// Mitsubishi GX Works2 project: BookEX6_48 Network   PLC: Q13UDV

// global labels: QPLCSpecial
VAR_GLOBAL
  sbGetTime AT SM213 : BOOL;
  sbOn AT SM400 : BOOL;
  sbOff AT SM401 : BOOL;
  sbOn1Time AT SM402 : BOOL;
  sbOff1Time AT SM403 : BOOL;
  sb5ms AT SM409 : BOOL;
  sdSwitch AT SD200 : INT;
  sdTime03 AT SD212 : INT;
  sdTime04 AT SD213 : INT;
  sdTime02 AT SD211 : INT;
  sdTime01 AT SD210 : INT;
  sdScanTime1 AT SD521 : INT;
  sdScanTimeMin1 AT SD525 : INT;
  sdScanTimeMin AT SD524 : INT;
  sdScanTimeMax1 AT SD527 : INT;
  sdScanTimeMax AT SD526 : INT;
  sbErrInfo2 AT SM16 : BOOL;
  sbErrInfo AT SM5 : BOOL;
  sbSelfError AT SM1 : BOOL;
  sbDiagError AT SM0 : BOOL;
  sbResetErr AT SM50 : BOOL;
  sbSetTime AT SM210 : BOOL;
  sbFuse AT SM60 : BOOL;
  sbOpError AT SM56 : BOOL;
  sbPowerDown AT SM53 : BOOL;
  sbBatLow AT SM52 : BOOL;
  sbBatLowL AT SM51 : BOOL;
  sbSTOP AT SM203 : BOOL;
  sbPAUSE AT SM204 : BOOL;
  sbNsec AT SM414 : BOOL;
  sb1000ms AT SM413 : BOOL;
  sb500ms AT SM412 : BOOL;
  sbNms AT SM415 : BOOL;
  sbUserClk4 AT SM424 : BOOL;
  sbUserClk3 AT SM423 : BOOL;
  sbUserClk2 AT SM422 : BOOL;
  sbUserClk1 AT SM421 : BOOL;
  sbUserClk0 AT SM420 : BOOL;
  sdBatLowL AT SD51 : INT;
  sdPLCErrInfo AT SD4 : INT;
  sdPLCErrDate2 AT SD3 : INT;
  sdPLCErrDate1 AT SD2 : INT;
  sdPLCErrDate0 AT SD1 : INT;
  sdPLCErrCode AT SD0 : INT;
  sdFuse AT SD60 : INT;
  sdPowerDown AT SD53 : INT;
  sdBatLow AT SD52 : INT;
  sdCPUSts AT SD203 : INT;
  sdLed AT SD201 : INT;
  sdScanTime AT SD520 : INT;
  sdCntNsec AT SD414 : INT;
  sdCnt1sec AT SD412 : INT;
  sdCntScan AT SD420 : INT;
  sdCntNms AT SD415 : INT;
  sb100ms AT SM411 : BOOL;
  sb50ms AT SM410 : BOOL;
  sdSckOpenComp AT SD1282 : WORD;
  sdSckOpenReq AT SD1284 : WORD;
  sdSckDataRx AT SD1286 : WORD;
  sdSckConn AT SD1288 : WORD;
END_VAR

// global labels: Network
VAR_GLOBAL
  aSendData1 AT D100 : ARRAY [0..4] OF INT;
  aiTxData AT D4000 : ARRAY [0..99] OF INT;
  aiRxData AT D4100 : ARRAY [0..99] OF INT;
  iOpenOK AT D3900 : INT;
  iOpenERR AT D3901 : INT;
  iSendOK AT D3902 : INT;
  iSendERR AT D3903 : INT;
  iCloseOK AT D3906 : INT;
  iCloseERR AT D3907 : INT;
  iRecvOK AT D3904 : INT;
  iRecvERR AT D3905 : INT;
  aiTxData2 AT D4200 : ARRAY [0..99] OF INT;
  aiRxData2 AT D4300 : ARRAY [0..99] OF INT;
  iOpenOK2 AT D3908 : INT;
  iOpenERR2 AT D3909 : INT;
  iSendOK2 AT D3910 : INT;
  iSendERR2 AT D3911 : INT;
  iRecvOK2 AT D3912 : INT;
  iRecvERR2 AT D3913 : INT;
  iCloseOK2 AT D3914 : INT;
  iCloseERR2 AT D3915 : INT;
  iEOpenComp AT D3916 : INT;
  iEOpenReq AT D3917 : INT;
  iERecvFlag AT D3918 : INT;
  iOpenCode AT D3919 : INT;
  iSendCode AT D3920 : INT;
  iRecvCode AT D3921 : INT;
  iCloseCode AT D3922 : INT;
  iOpenCode2 AT D3923 : INT;
  iSendCode2 AT D3924 : INT;
  iRecvCode2 AT D3925 : INT;
  iCloseCode2 AT D3926 : INT;
  aRecvData1 AT D105 : ARRAY [0..4] OF INT;
  aSendData2 AT D110 : ARRAY [0..4] OF INT;
  aRecvData2 AT D115 : ARRAY [0..4] OF INT;
  aSendData3 AT D120 : ARRAY [0..4] OF INT;
  aRecvData3 AT D125 : ARRAY [0..4] OF INT;
  aRdata AT D140 : ARRAY [0..9] OF INT;
  aSLMPDataTx AT D150 : ARRAY [0..9] OF WORD;
  aSLMPDataRx AT D160 : ARRAY [0..9] OF WORD;
END_VAR

// global labels: Global
VAR_GLOBAL
  bVar0 AT M5000 : BOOL;
  abArray0 AT M5010 : ARRAY [0..49] OF BOOL;
  sStr0 AT D5000 : STRING[199];
  sStr1 AT D5100 : STRING[199];
  sStr2 AT D5200 : STRING[199];
  sStr3 AT D5300 : STRING[199];
  sStr4 AT D5400 : STRING[199];
  sStr5 AT D5500 : STRING[199];
  sStr6 AT D5600 : STRING[199];
  sStr7 AT D5700 : STRING[199];
  sStr8 AT D5800 : STRING[199];
  sStr9 AT D5900 : STRING[199];
  iVar0 AT D4500 : INT;
  iVar1 AT D4501 : INT;
  iVar2 AT D4502 : INT;
  iVar3 AT D4503 : INT;
  iVar4 AT D4504 : INT;
  iVar5 AT D4505 : INT;
  iVar6 AT D4506 : INT;
  iVar7 AT D4507 : INT;
  iVar8 AT D4508 : INT;
  iVar9 AT D4509 : INT;
  dVar0 AT D4510 : DINT;
  dVar1 AT D4512 : DINT;
  dVar2 AT D4514 : DINT;
  dVar3 AT D4516 : DINT;
  dVar4 AT D4518 : DINT;
  dVar5 AT D4520 : DINT;
  dVar6 AT D4522 : DINT;
  dVar7 AT D4524 : DINT;
  dVar8 AT D4526 : DINT;
  dVar9 AT D4528 : DINT;
  wVar0 AT D4530 : WORD;
  wVar1 AT D4531 : WORD;
  wVar2 AT D4532 : WORD;
  wVar3 AT D4533 : WORD;
  wVar4 AT D4534 : WORD;
  wVar5 AT D4535 : WORD;
  wVar6 AT D4536 : WORD;
  wVar7 AT D4537 : WORD;
  wVar8 AT D4538 : WORD;
  wVar9 AT D4539 : WORD;
  dwVar0 AT D4540 : DWORD;
  dwVar1 AT D4542 : DWORD;
  dwVar2 AT D4544 : DWORD;
  dwVar3 AT D4546 : DWORD;
  dwVar4 AT D4548 : DWORD;
  dwVar5 AT D4550 : DWORD;
  dwVar6 AT D4552 : DWORD;
  dwVar7 AT D4554 : DWORD;
  dwVar8 AT D4556 : DWORD;
  dwVar9 AT D4558 : DWORD;
  fsVar0 AT D4560 : REAL;
  fsVar1 AT D4562 : REAL;
  fsVar2 AT D4564 : REAL;
  fsVar3 AT D4566 : REAL;
  fsVar4 AT D4568 : REAL;
  fsVar5 AT D4570 : REAL;
  fsVar6 AT D4572 : REAL;
  fsVar7 AT D4574 : REAL;
  fsVar8 AT D4576 : REAL;
  fsVar9 AT D4578 : REAL;
  fdVar0 AT D4580 : LREAL;
  tTime0 AT D4620 : TIME;
  tTime1 AT D4622 : TIME;
  tTime2 AT D4624 : TIME;
  tTime3 AT D4626 : TIME;
  tTime4 AT D4628 : TIME;
  tTime5 AT D4630 : TIME;
  tTime6 AT D4632 : TIME;
  tTime7 AT D4634 : TIME;
  tTime8 AT D4636 : TIME;
  tTime9 AT D4638 : TIME;
  tTime10 AT D4640 : TIME;
  bVar1 AT M5001 : BOOL;
  bVar2 AT M5002 : BOOL;
  bVar3 AT M5003 : BOOL;
  bVar4 AT M5004 : BOOL;
  bVar5 AT M5005 : BOOL;
  bVar6 AT M5006 : BOOL;
  bVar7 AT M5007 : BOOL;
  bVar8 AT M5008 : BOOL;
  bVar9 AT M5009 : BOOL;
  abArray1 AT M5060 : ARRAY [0..49] OF BOOL;
  abArray2 AT M5110 : ARRAY [0..49] OF BOOL;
  abArray3 AT M5160 : ARRAY [0..49] OF BOOL;
  abArray4 AT M5210 : ARRAY [0..49] OF BOOL;
  abArray5 AT M5260 : ARRAY [0..49] OF BOOL;
  abArray6 AT M5310 : ARRAY [0..49] OF BOOL;
  abArray7 AT M5360 : ARRAY [0..49] OF BOOL;
  abArray8 AT M5410 : ARRAY [0..49] OF BOOL;
  abArray9 AT M5460 : ARRAY [0..49] OF BOOL;
  fdVar1 AT D4584 : LREAL;
  fdVar2 AT D4588 : LREAL;
  fdVar3 AT D4592 : LREAL;
  fdVar4 AT D4596 : LREAL;
  fdVar5 AT D4600 : LREAL;
  fdVar6 AT D4604 : LREAL;
  fdVar7 AT D4608 : LREAL;
  fdVar8 AT D4612 : LREAL;
  fdVar9 AT D4616 : LREAL;
  afsPen0 AT D2000 : ARRAY [0..499] OF REAL;
  afsPen1 AT D3000 : ARRAY [0..499] OF REAL;
END_VAR
// user libraries (not included): HMI

PROGRAM ExEpasCact
VAR
  bOpenReqC : BOOL;
  bOpenOkC : BOOL;
  bOpenErrC : BOOL;
  abOpenResC : ARRAY [0..1] OF BOOL;
  acOpenData : ARRAY [0..9] OF INT;
  bSendReqC : BOOL;
  bSendOkC : BOOL;
  bSendErrC : BOOL;
  abSendResC : ARRAY [0..1] OF BOOL;
  acSendDataC : ARRAY [0..1] OF INT;
  bRecvOkC : BOOL;
  bRecvErrC : BOOL;
  abRecvResC : ARRAY [0..1] OF BOOL;
  bCloseReq : BOOL;
  bCloseOkC : BOOL;
  bCloseErrC : BOOL;
  abCloseResC : ARRAY [0..1] OF BOOL;
  acCloseData : ARRAY [0..1] OF INT;
  CntSend1 : INT;
  CntSend2 : INT;
  CntRecv1 : INT;
  CntRecv2 : INT;
  Mov4INT_1 : Mov4INT;
  Mov8INT_1 : Mov8INT;
  acRdCtrl : ARRAY [0..9] OF INT;
  Mov4INT_2 : Mov4INT;
  bOpenReqE : BOOL;
  bOpenOkE : BOOL;
  bOpenErrE : BOOL;
  abOpenResE : ARRAY [0..1] OF BOOL;
  bSendErrE : BOOL;
  bSendOkE : BOOL;
  bSendReqE : BOOL;
  abSendResE : ARRAY [0..1] OF BOOL;
  abRecvResE : ARRAY [0..1] OF BOOL;
  bRecvErrE : BOOL;
  bRecvOkE : BOOL;
  abCloseResE : ARRAY [0..1] OF BOOL;
  bCloseErrE : BOOL;
  bCloseOkE : BOOL;
  acSendDataE : ARRAY [0..1] OF INT;
  acRecvDataC : ARRAY [0..1] OF INT;
  acRecvDataE : ARRAY [0..1] OF INT;
  Word2Bit8_1 : Word2Bit8;
  Word2Bit8_2 : Word2Bit8;
  Word2Bit8_3 : Word2Bit8;
  Word2Bit8_4 : Word2Bit8;
  Word2Bit8_5 : Word2Bit8;
  Word2Bit8_6 : Word2Bit8;
  ErrCodeSC : INT;
  ErrCodeSE : INT;
  Mov4INT_3 : Mov4INT;
  bChangeReqC : BOOL;
  Mov4INT_4 : Mov4INT;
  acRmodeData : ARRAY [0..3] OF INT;
  TON_1 : TON;
  CntRecvErr1 : INT;
  CntRecvErr2 : INT;
  TON_2 : TON;
  ErrCodeRC : INT;
  ErrCodeRE : INT;
  bModeReq : BOOL;
  acRdata : ARRAY [0..1] OF INT;
END_VAR
(* structured ladder/FBD written out as ST: instructions are called as NAME(EN, inputs, outputs); _pN, _eN, _tN stand for wires *)
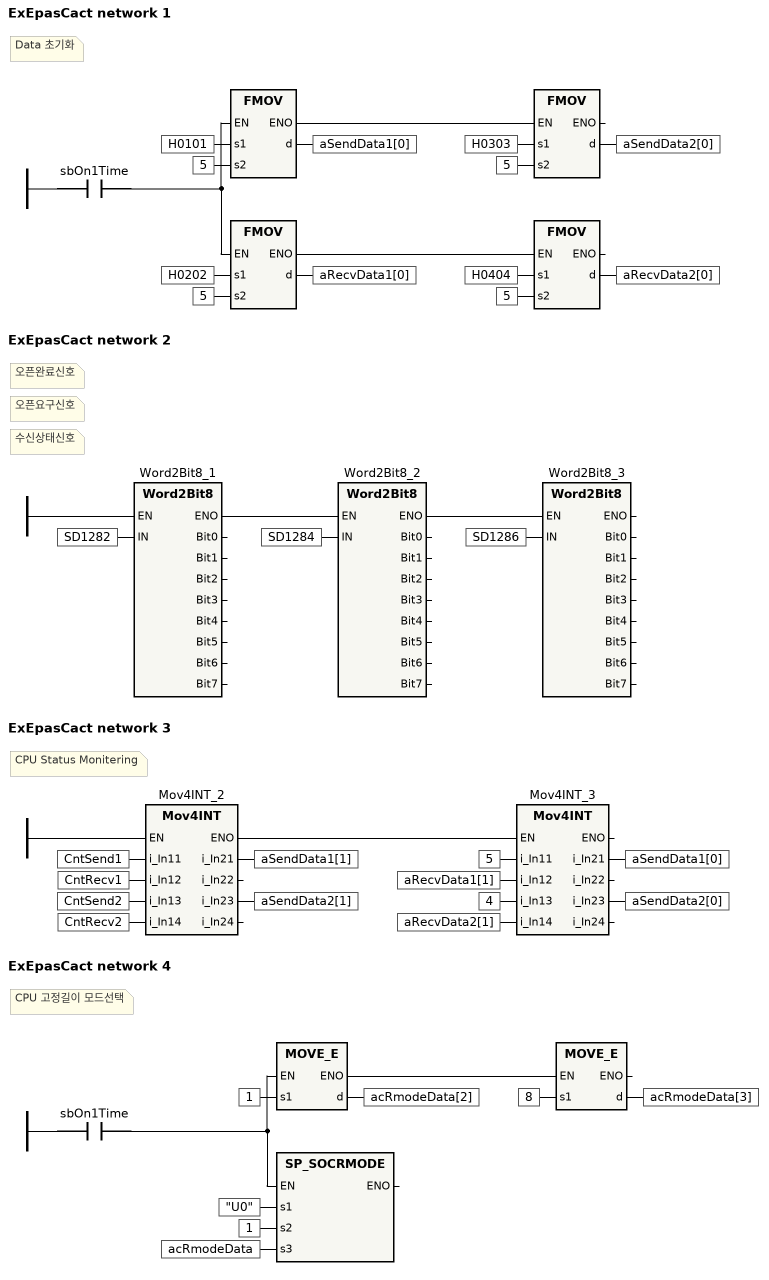
(* network 1 *)
(* Data 초기화 *)
_e1 := FMOV(sbOn1Time, H0101, 5, aSendData1[0]);
FMOV(_e1, H0303, 5, aSendData2[0]);
_e2 := FMOV(sbOn1Time, H0202, 5, aRecvData1[0]);
FMOV(_e2, H0404, 5, aRecvData2[0]);
(* network 2 *)
(* 오픈완료신호 *)
(* 오픈요구신호 *)
(* 수신상태신호 *)
Word2Bit8_1(EN := TRUE, IN := SD1282);
Word2Bit8_2(EN := Word2Bit8_1.ENO, IN := SD1284);
Word2Bit8_3(EN := Word2Bit8_2.ENO, IN := SD1286);
(* network 3 *)
(* CPU Status Monitering *)
Mov4INT_2(EN := TRUE, i_In11 := CntSend1, i_In12 := CntRecv1, i_In13 := CntSend2, i_In14 := CntRecv2, i_In21 => aSendData1[1], i_In23 => aSendData2[1]);
Mov4INT_3(EN := Mov4INT_2.ENO, i_In11 := 5, i_In12 := aRecvData1[1], i_In13 := 4, i_In14 := aRecvData2[1], i_In21 => aSendData1[0], i_In23 => aSendData2[0]);
(* network 4 *)
(* CPU 고정길이 모드선택 *)
_e1 := MOVE_E(sbOn1Time, 1, acRmodeData[2]);
MOVE_E(_e1, 8, acRmodeData[3]);
SP_SOCRMODE(sbOn1Time, "U0", 1, acRmodeData);
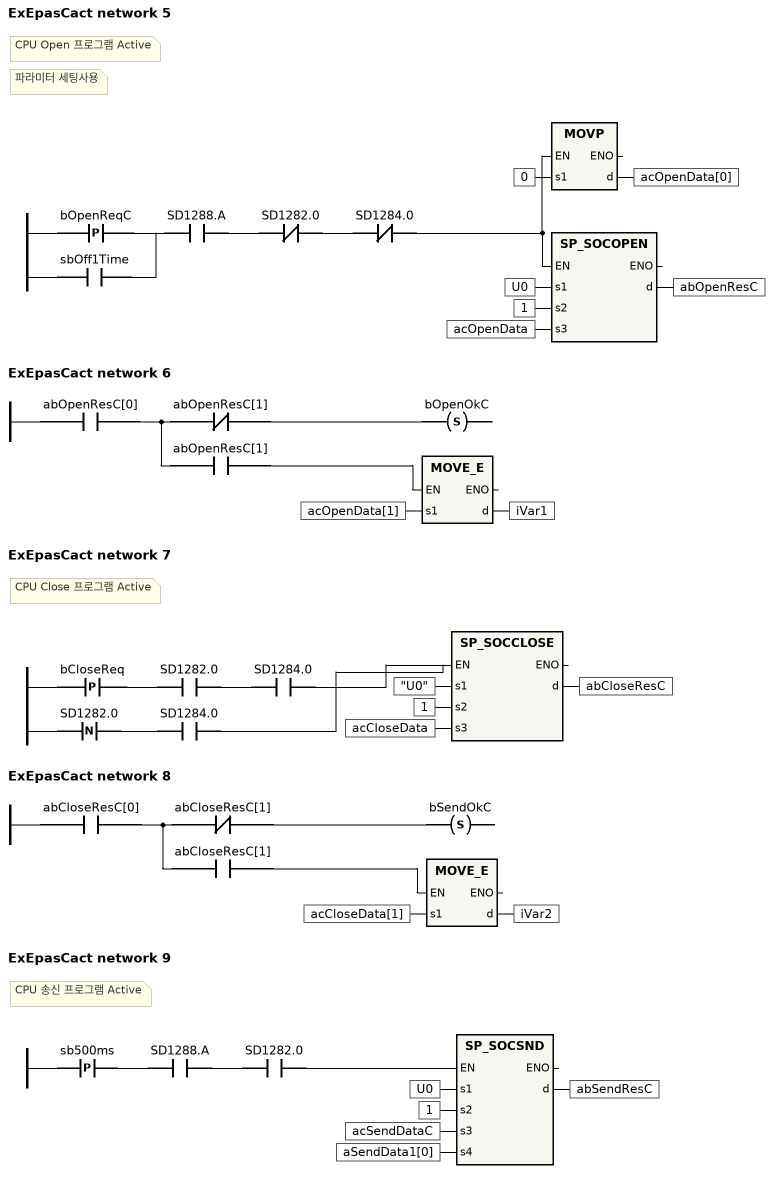
(* network 5 *)
(* CPU Open 프로그램 Active *)
(* 파라미터 세팅사용 *)
_p1 := (((LDP(TRUE, bOpenReqC) OR sbOff1Time) AND SD1288.A) AND NOT SD1282.0) AND NOT SD1284.0;
MOVP(_p1, 0, acOpenData[0]);
SP_SOCOPEN(_p1, U0, 1, acOpenData, abOpenResC);
(* network 6 *)
SET(abOpenResC[0] AND NOT abOpenResC[1], bOpenOkC);
MOVE_E(abOpenResC[0] AND abOpenResC[1], acOpenData[1], iVar1);
(* network 7 *)
(* CPU Close 프로그램 Active *)
SP_SOCCLOSE((LDP(TRUE, bCloseReq) AND SD1282.0 AND SD1284.0) OR (LDF(TRUE, SD1282.0) AND SD1284.0), "U0", 1, acCloseData, abCloseResC);
(* network 8 *)
SET(abCloseResC[0] AND NOT abCloseResC[1], bSendOkC);
MOVE_E(abCloseResC[0] AND abCloseResC[1], acCloseData[1], iVar2);
(* network 9 *)
(* CPU 송신 프로그램 Active *)
SP_SOCSND(LDP(TRUE, sb500ms) AND SD1288.A AND SD1282.0, U0, 1, acSendDataC, aSendData1[0], abSendResC);
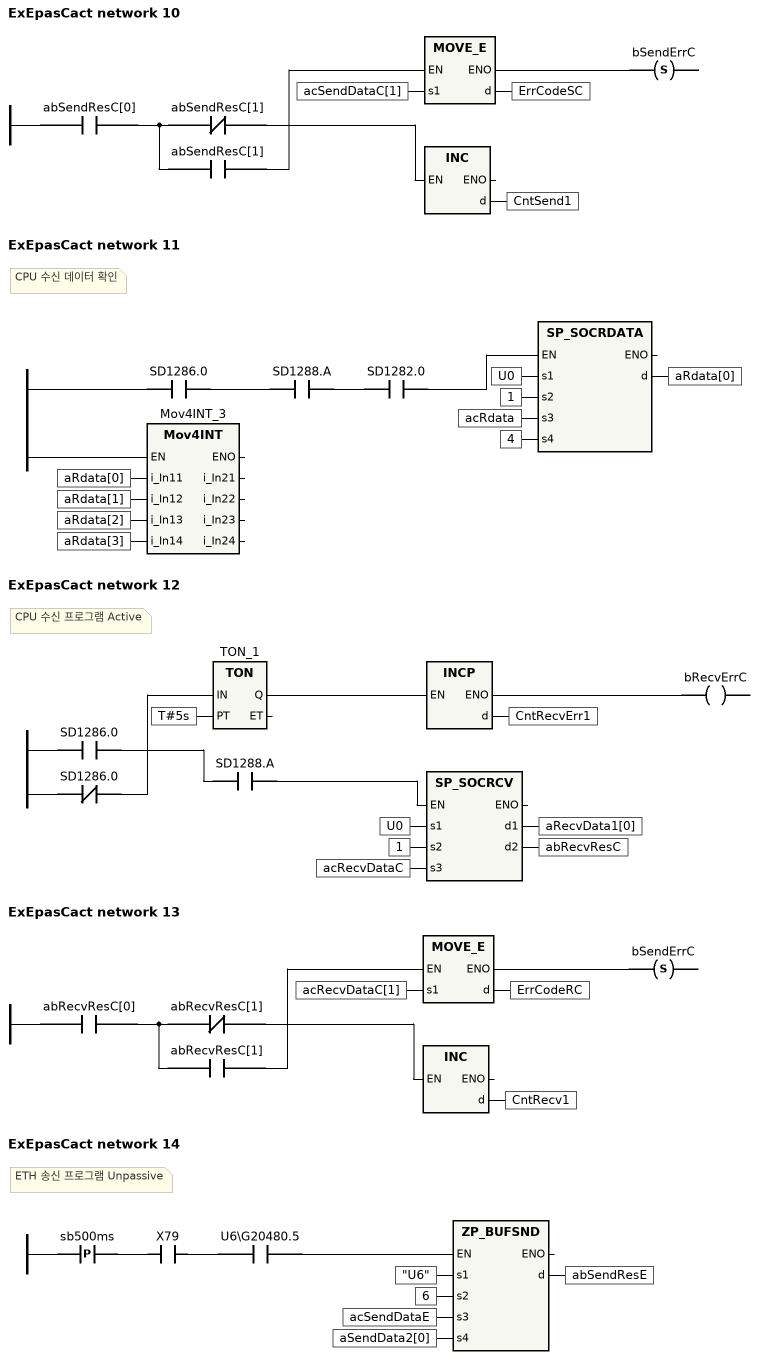
(* network 10 *)
INC(abSendResC[0] AND NOT abSendResC[1], CntSend1);
_e1 := MOVE_E(abSendResC[0] AND abSendResC[1], acSendDataC[1], ErrCodeSC);
SET(_e1, bSendErrC);
(* network 11 *)
(* CPU 수신 데이터 확인 *)
SP_SOCRDATA(SD1286.0 AND SD1288.A AND SD1282.0, U0, 1, acRdata, 4, aRdata[0]);
Mov4INT_3(EN := TRUE, i_In11 := aRdata[0], i_In12 := aRdata[1], i_In13 := aRdata[2], i_In14 := aRdata[3]);
(* network 12 *)
(* CPU 수신 프로그램 Active *)
SP_SOCRCV(SD1286.0 AND SD1288.A, U0, 1, acRecvDataC, aRecvData1[0], abRecvResC);
TON_1(IN := NOT SD1286.0, PT := T#5s);
_e1 := INCP(TON_1.Q, CntRecvErr1);
bRecvErrC := _e1;
(* network 13 *)
INC(abRecvResC[0] AND NOT abRecvResC[1], CntRecv1);
_e1 := MOVE_E(abRecvResC[0] AND abRecvResC[1], acRecvDataC[1], ErrCodeRC);
SET(_e1, bSendErrC);
(* network 14 *)
(* ETH 송신 프로그램 Unpassive *)
ZP_BUFSND(LDP(TRUE, sb500ms) AND X79 AND U6\G20480.5, "U6", 6, acSendDataE, aSendData2[0], abSendResE);
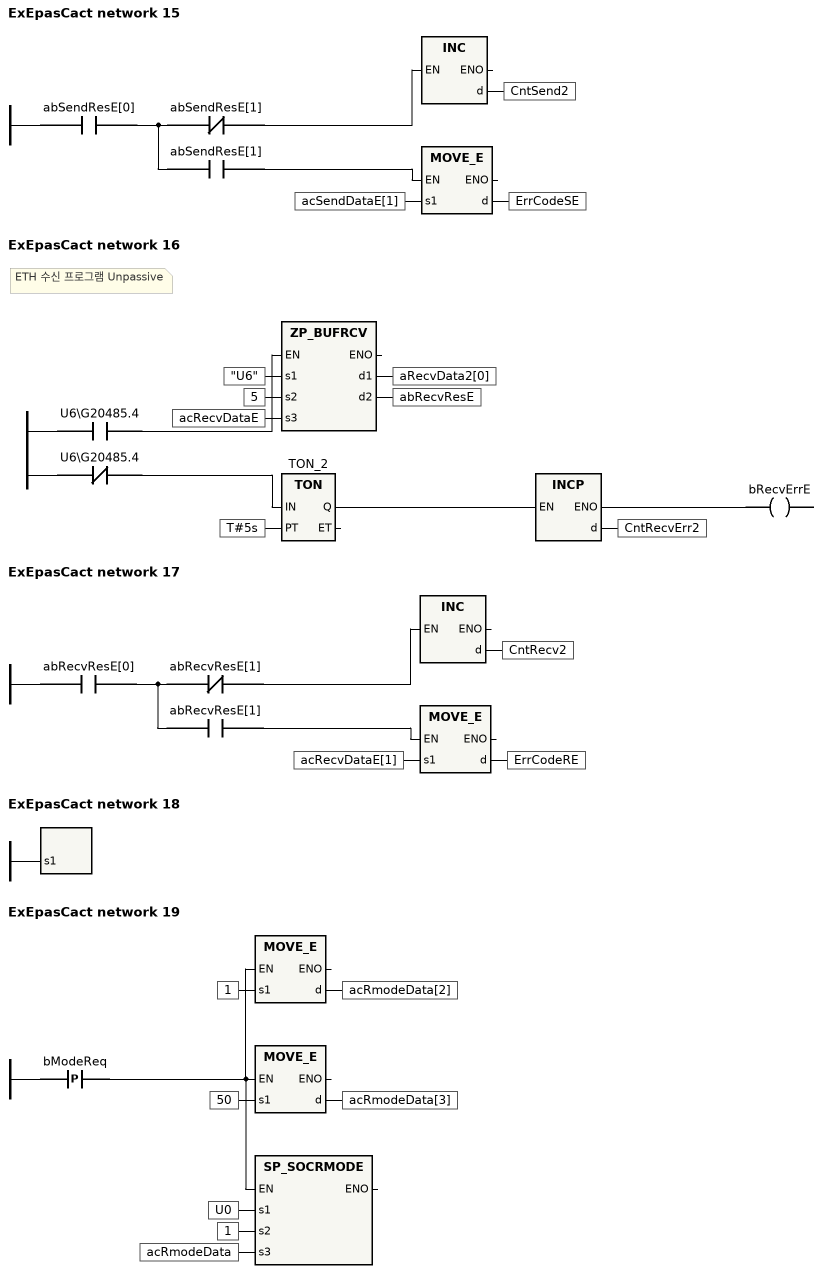
(* network 15 *)
INC(abSendResE[0] AND NOT abSendResE[1], CntSend2);
MOVE_E(abSendResE[0] AND abSendResE[1], acSendDataE[1], ErrCodeSE);
(* network 16 *)
(* ETH 수신 프로그램 Unpassive *)
ZP_BUFRCV(U6\G20485.4, "U6", 5, acRecvDataE, aRecvData2[0], abRecvResE);
TON_2(IN := NOT U6\G20485.4, PT := T#5s);
_e1 := INCP(TON_2.Q, CntRecvErr2);
bRecvErrE := _e1;
(* network 17 *)
INC(abRecvResE[0] AND NOT abRecvResE[1], CntRecv2);
MOVE_E(abRecvResE[0] AND abRecvResE[1], acRecvDataE[1], ErrCodeRE);
(* network 18 *)
(* element kind 10  <- TRUE *)
(* network 19 *)
_p1 := LDP(TRUE, bModeReq);
MOVE_E(_p1, 1, acRmodeData[2]);
MOVE_E(_p1, 50, acRmodeData[3]);
SP_SOCRMODE(_p1, U0, 1, acRmodeData);
END_PROGRAM

PROGRAM xEx_ethOPENact
(* structured ladder/FBD written out as ST: instructions are called as NAME(EN, inputs, outputs); _pN, _eN, _tN stand for wires *)
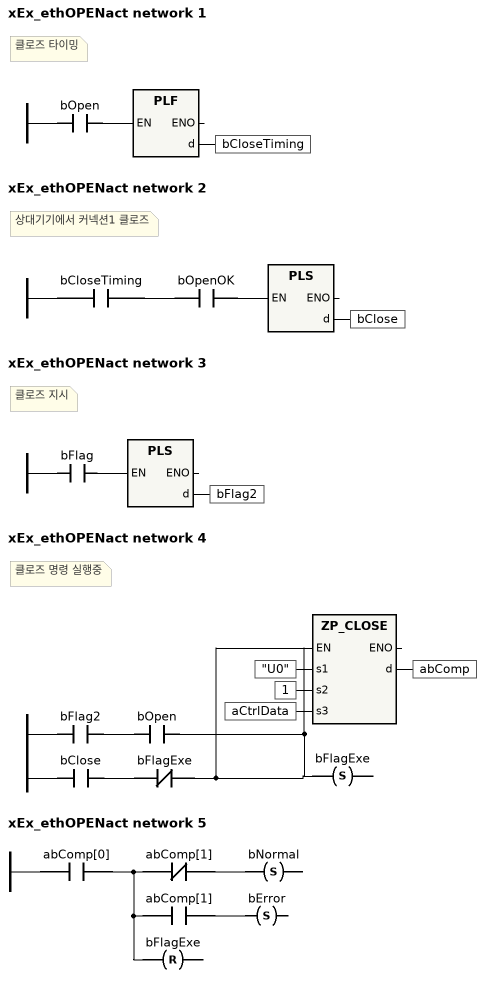
(* network 1 *)
(* 클로즈 타이밍 *)
PLF(bOpen, bCloseTiming);
(* network 2 *)
(* 상대기기에서 커넥션1 클로즈 *)
PLS(bCloseTiming AND bOpenOK, bClose);
(* network 3 *)
(* 클로즈 지시 *)
PLS(bFlag, bFlag2);
(* network 4 *)
(* 클로즈 명령 실행중 *)
_p1 := (bFlag2 AND bOpen) OR (bClose AND NOT bFlagExe);
ZP_CLOSE(_p1, "U0", 1, aCtrlData, abComp);
SET(_p1, bFlagExe);
(* network 5 *)
SET(abComp[0] AND NOT abComp[1], bNormal);
SET(abComp[0] AND abComp[1], bError);
RST(abComp[0], bFlagExe);
END_PROGRAM

PROGRAM xEx_OPENact
VAR
  Mov4INT_1 : Mov4INT;
  abOpenComp : ARRAY [0..1] OF BOOL;
  acOpenData : ARRAY [0..9] OF INT;
  abSendComp : ARRAY [0..1] OF BOOL;
  acSendData : ARRAY [0..1] OF INT;
  abRecvComp : ARRAY [0..1] OF BOOL;
  acRecvData : ARRAY [0..1] OF INT;
  abCloseComp : ARRAY [0..1] OF BOOL;
  acCloseData : ARRAY [0..1] OF INT;
  Word2Bit_1 : Word2Bit;
  Word2Bit_2 : Word2Bit;
  Word2Bit_3 : Word2Bit;
  abOpen : ARRAY [1..16] OF BOOL;
  abReq : ARRAY [1..16] OF BOOL;
  abRecv : ARRAY [1..16] OF BOOL;
  abOpenComp2 : ARRAY [0..1] OF BOOL;
  acOpenData2 : ARRAY [0..9] OF INT;
  abSendComp2 : ARRAY [0..1] OF BOOL;
  acSendData2 : ARRAY [0..1] OF INT;
  abRecvComp2 : ARRAY [0..1] OF BOOL;
  acRecvData2 : ARRAY [0..1] OF INT;
  abCloseComp2 : ARRAY [0..1] OF BOOL;
  acCloseData2 : ARRAY [0..1] OF INT;
  Mov4INT_2 : Mov4INT;
  Word2Bit_4 : Word2Bit;
  Word2Bit_5 : Word2Bit;
  Word2Bit_6 : Word2Bit;
  abRecv2 : ARRAY [1..16] OF BOOL;
  abOpen2 : ARRAY [1..16] OF BOOL;
  abReq2 : ARRAY [1..16] OF BOOL;
  bRecvOK : BOOL;
END_VAR
(* structured ladder/FBD written out as ST: instructions are called as NAME(EN, inputs, outputs); _pN, _eN, _tN stand for wires *)
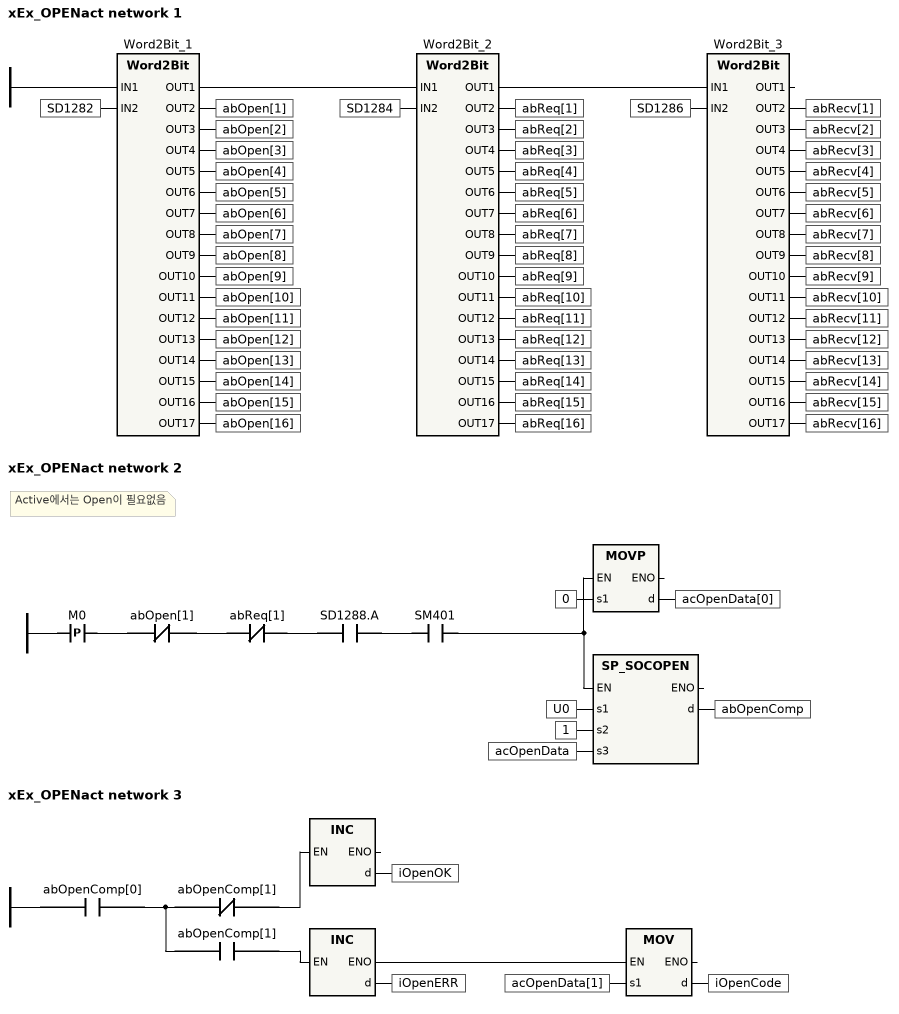
(* network 1 *)
Word2Bit_1(IN1 := TRUE, IN2 := SD1282, OUT2 => abOpen[1], OUT3 => abOpen[2], OUT4 => abOpen[3], OUT5 => abOpen[4], OUT6 => abOpen[5], OUT7 => abOpen[6], OUT8 => abOpen[7], OUT9 => abOpen[8], OUT10 => abOpen[9], OUT11 => abOpen[10], OUT12 => abOpen[11], OUT13 => abOpen[12], OUT14 => abOpen[13], OUT15 => abOpen[14], OUT16 => abOpen[15], OUT17 => abOpen[16]);
Word2Bit_2(IN1 := Word2Bit_1.OUT1, IN2 := SD1284, OUT2 => abReq[1], OUT3 => abReq[2], OUT4 => abReq[3], OUT5 => abReq[4], OUT6 => abReq[5], OUT7 => abReq[6], OUT8 => abReq[7], OUT9 => abReq[8], OUT10 => abReq[9], OUT11 => abReq[10], OUT12 => abReq[11], OUT13 => abReq[12], OUT14 => abReq[13], OUT15 => abReq[14], OUT16 => abReq[15], OUT17 => abReq[16]);
Word2Bit_3(IN1 := Word2Bit_2.OUT1, IN2 := SD1286, OUT2 => abRecv[1], OUT3 => abRecv[2], OUT4 => abRecv[3], OUT5 => abRecv[4], OUT6 => abRecv[5], OUT7 => abRecv[6], OUT8 => abRecv[7], OUT9 => abRecv[8], OUT10 => abRecv[9], OUT11 => abRecv[10], OUT12 => abRecv[11], OUT13 => abRecv[12], OUT14 => abRecv[13], OUT15 => abRecv[14], OUT16 => abRecv[15], OUT17 => abRecv[16]);
(* network 2 *)
(* Active에서는 Open이 필요없음 *)
_p1 := LDP(TRUE, M0) AND NOT abOpen[1] AND NOT abReq[1] AND SD1288.A AND SM401;
MOVP(_p1, 0, acOpenData[0]);
SP_SOCOPEN(_p1, U0, 1, acOpenData, abOpenComp);
(* network 3 *)
INC(abOpenComp[0] AND NOT abOpenComp[1], iOpenOK);
_e1 := INC(abOpenComp[0] AND abOpenComp[1], iOpenERR);
MOV(_e1, acOpenData[1], iOpenCode);
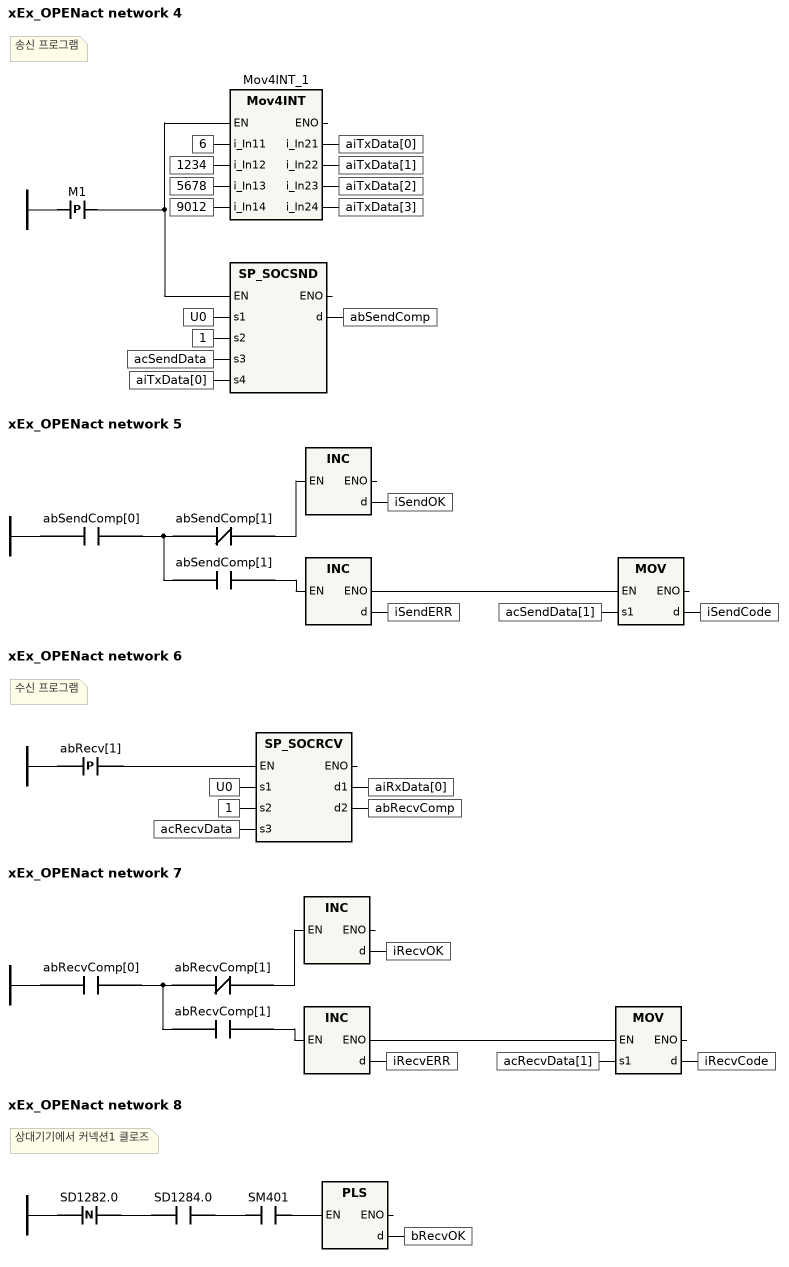
(* network 4 *)
(* 송신 프로그램 *)
_p1 := LDP(TRUE, M1);
Mov4INT_1(EN := _p1, i_In11 := 6, i_In12 := 1234, i_In13 := 5678, i_In14 := 9012, i_In21 => aiTxData[0], i_In22 => aiTxData[1], i_In23 => aiTxData[2], i_In24 => aiTxData[3]);
SP_SOCSND(_p1, U0, 1, acSendData, aiTxData[0], abSendComp);
(* network 5 *)
INC(abSendComp[0] AND NOT abSendComp[1], iSendOK);
_e1 := INC(abSendComp[0] AND abSendComp[1], iSendERR);
MOV(_e1, acSendData[1], iSendCode);
(* network 6 *)
(* 수신 프로그램 *)
SP_SOCRCV(LDP(TRUE, abRecv[1]), U0, 1, acRecvData, aiRxData[0], abRecvComp);
(* network 7 *)
INC(abRecvComp[0] AND NOT abRecvComp[1], iRecvOK);
_e1 := INC(abRecvComp[0] AND abRecvComp[1], iRecvERR);
MOV(_e1, acRecvData[1], iRecvCode);
(* network 8 *)
(* 상대기기에서 커넥션1 클로즈 *)
PLS(LDF(TRUE, SD1282.0) AND SD1284.0 AND SM401, bRecvOK);
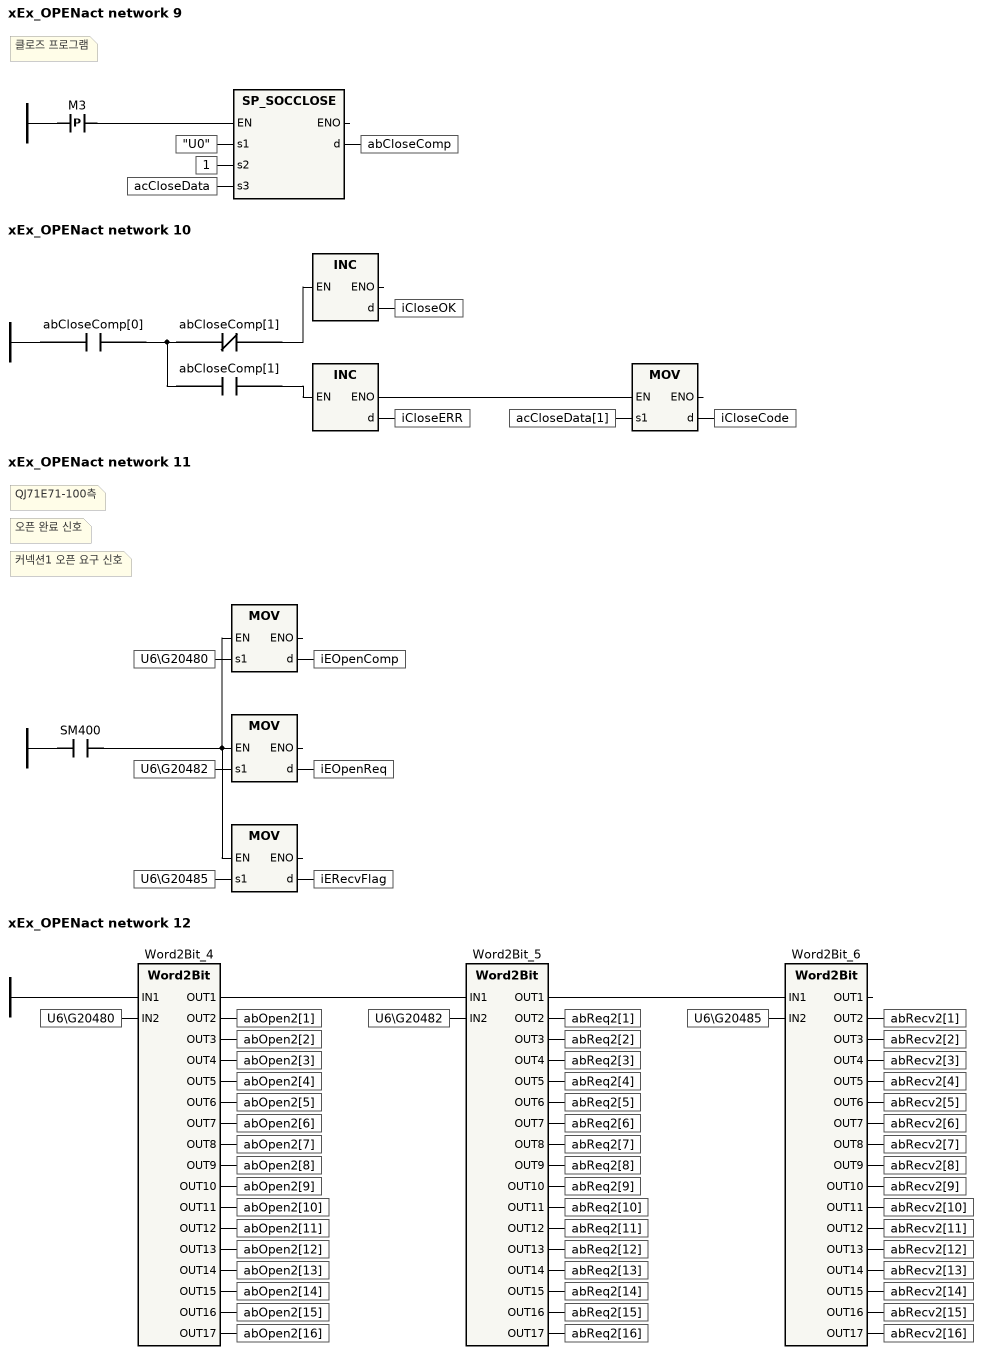
(* network 9 *)
(* 클로즈 프로그램 *)
SP_SOCCLOSE(LDP(TRUE, M3), "U0", 1, acCloseData, abCloseComp);
(* network 10 *)
INC(abCloseComp[0] AND NOT abCloseComp[1], iCloseOK);
_e1 := INC(abCloseComp[0] AND abCloseComp[1], iCloseERR);
MOV(_e1, acCloseData[1], iCloseCode);
(* network 11 *)
(* QJ71E71-100측 *)
(* 오픈 완료 신호 *)
(* 커넥션1 오픈 요구 신호 *)
MOV(SM400, U6\G20480, iEOpenComp);
MOV(SM400, U6\G20482, iEOpenReq);
MOV(SM400, U6\G20485, iERecvFlag);
(* network 12 *)
Word2Bit_4(IN1 := TRUE, IN2 := U6\G20480, OUT2 => abOpen2[1], OUT3 => abOpen2[2], OUT4 => abOpen2[3], OUT5 => abOpen2[4], OUT6 => abOpen2[5], OUT7 => abOpen2[6], OUT8 => abOpen2[7], OUT9 => abOpen2[8], OUT10 => abOpen2[9], OUT11 => abOpen2[10], OUT12 => abOpen2[11], OUT13 => abOpen2[12], OUT14 => abOpen2[13], OUT15 => abOpen2[14], OUT16 => abOpen2[15], OUT17 => abOpen2[16]);
Word2Bit_5(IN1 := Word2Bit_4.OUT1, IN2 := U6\G20482, OUT2 => abReq2[1], OUT3 => abReq2[2], OUT4 => abReq2[3], OUT5 => abReq2[4], OUT6 => abReq2[5], OUT7 => abReq2[6], OUT8 => abReq2[7], OUT9 => abReq2[8], OUT10 => abReq2[9], OUT11 => abReq2[10], OUT12 => abReq2[11], OUT13 => abReq2[12], OUT14 => abReq2[13], OUT15 => abReq2[14], OUT16 => abReq2[15], OUT17 => abReq2[16]);
Word2Bit_6(IN1 := Word2Bit_5.OUT1, IN2 := U6\G20485, OUT2 => abRecv2[1], OUT3 => abRecv2[2], OUT4 => abRecv2[3], OUT5 => abRecv2[4], OUT6 => abRecv2[5], OUT7 => abRecv2[6], OUT8 => abRecv2[7], OUT9 => abRecv2[8], OUT10 => abRecv2[9], OUT11 => abRecv2[10], OUT12 => abRecv2[11], OUT13 => abRecv2[12], OUT14 => abRecv2[13], OUT15 => abRecv2[14], OUT16 => abRecv2[15], OUT17 => abRecv2[16]);
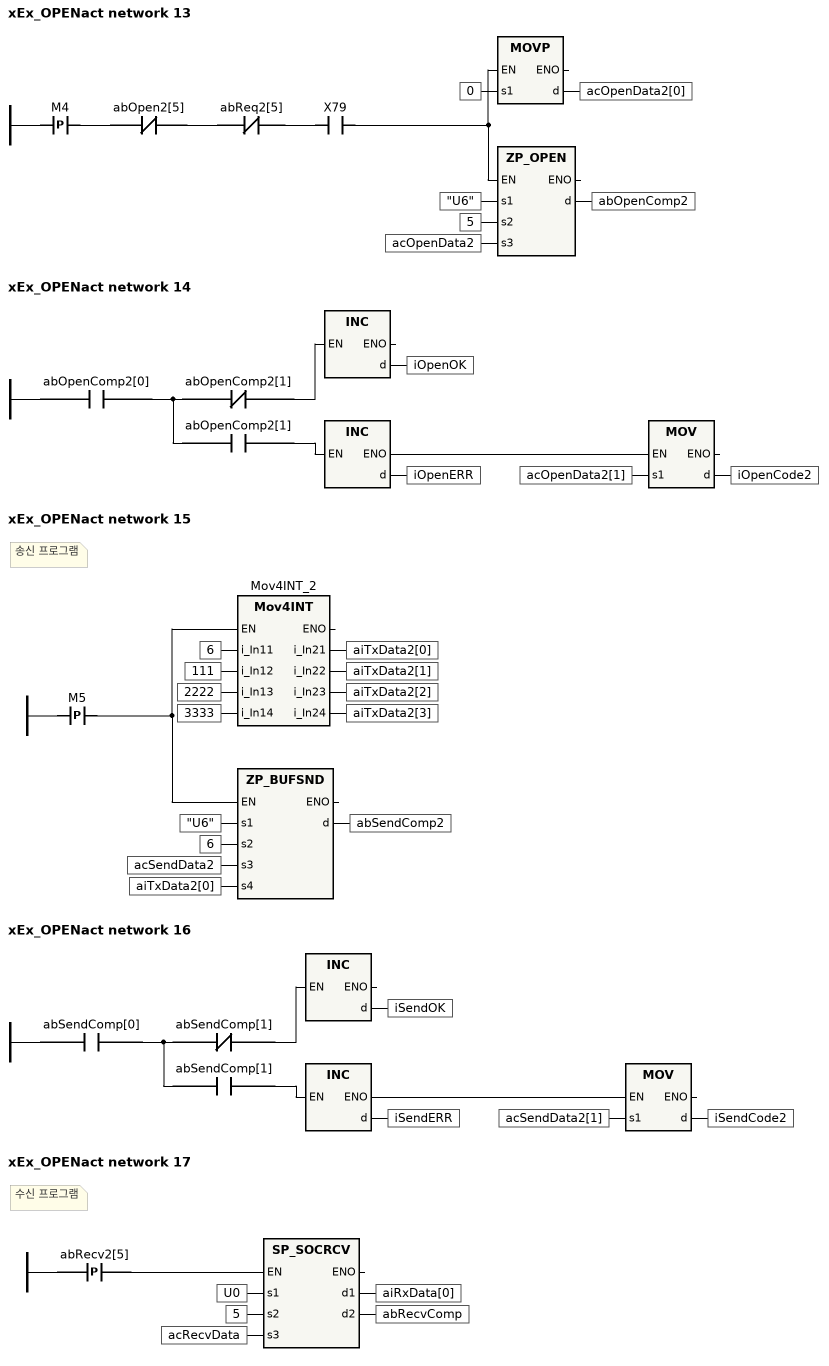
(* network 13 *)
_p1 := LDP(TRUE, M4) AND NOT abOpen2[5] AND NOT abReq2[5] AND X79;
MOVP(_p1, 0, acOpenData2[0]);
ZP_OPEN(_p1, "U6", 5, acOpenData2, abOpenComp2);
(* network 14 *)
INC(abOpenComp2[0] AND NOT abOpenComp2[1], iOpenOK);
_e1 := INC(abOpenComp2[0] AND abOpenComp2[1], iOpenERR);
MOV(_e1, acOpenData2[1], iOpenCode2);
(* network 15 *)
(* 송신 프로그램 *)
_p1 := LDP(TRUE, M5);
Mov4INT_2(EN := _p1, i_In11 := 6, i_In12 := 111, i_In13 := 2222, i_In14 := 3333, i_In21 => aiTxData2[0], i_In22 => aiTxData2[1], i_In23 => aiTxData2[2], i_In24 => aiTxData2[3]);
ZP_BUFSND(_p1, "U6", 6, acSendData2, aiTxData2[0], abSendComp2);
(* network 16 *)
INC(abSendComp[0] AND NOT abSendComp[1], iSendOK);
_e1 := INC(abSendComp[0] AND abSendComp[1], iSendERR);
MOV(_e1, acSendData2[1], iSendCode2);
(* network 17 *)
(* 수신 프로그램 *)
SP_SOCRCV(LDP(TRUE, abRecv2[5]), U0, 5, acRecvData, aiRxData[0], abRecvComp);
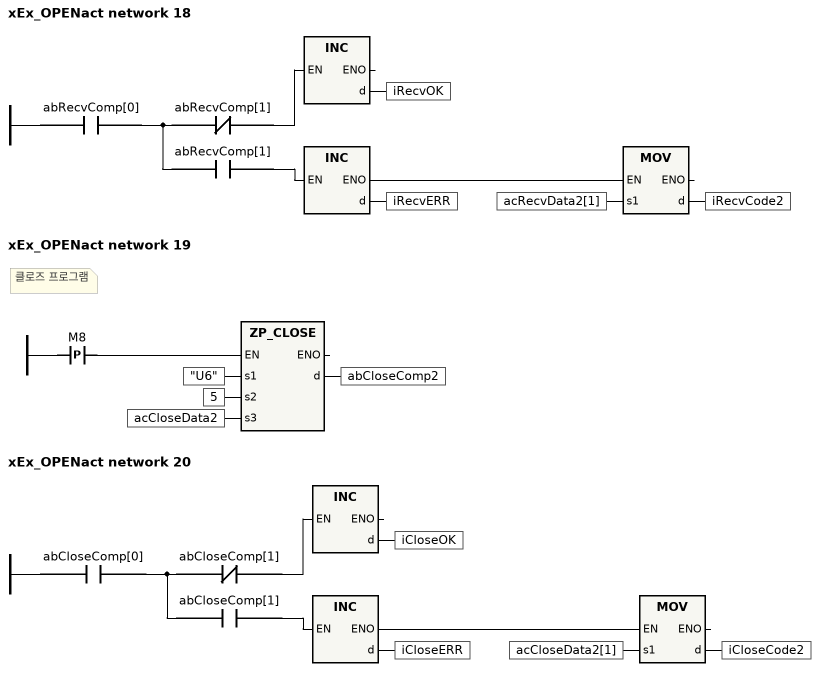
(* network 18 *)
INC(abRecvComp[0] AND NOT abRecvComp[1], iRecvOK);
_e1 := INC(abRecvComp[0] AND abRecvComp[1], iRecvERR);
MOV(_e1, acRecvData2[1], iRecvCode2);
(* network 19 *)
(* 클로즈 프로그램 *)
ZP_CLOSE(LDP(TRUE, M8), "U6", 5, acCloseData2, abCloseComp2);
(* network 20 *)
INC(abCloseComp[0] AND NOT abCloseComp[1], iCloseOK);
_e1 := INC(abCloseComp[0] AND abCloseComp[1], iCloseERR);
MOV(_e1, acCloseData2[1], iCloseCode2);
END_PROGRAM

PROGRAM ExBUFRCV
(* structured ladder/FBD written out as ST: instructions are called as NAME(EN, inputs, outputs); _pN, _eN, _tN stand for wires *)
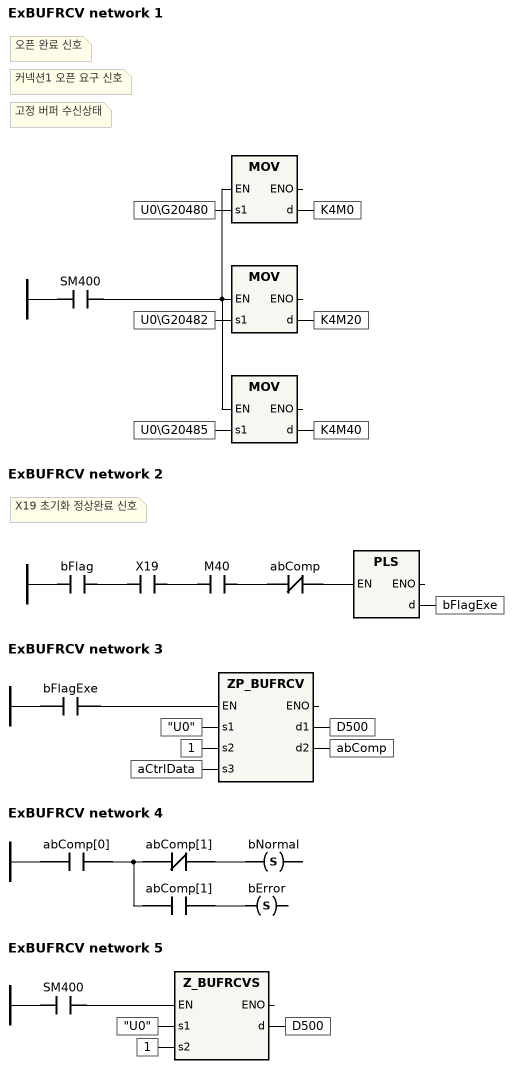
(* network 1 *)
(* 오픈 완료 신호 *)
(* 커넥션1 오픈 요구 신호 *)
(* 고정 버퍼 수신상태 *)
MOV(SM400, U0\G20480, K4M0);
MOV(SM400, U0\G20482, K4M20);
MOV(SM400, U0\G20485, K4M40);
(* network 2 *)
(* X19 초기화 정상완료 신호 *)
PLS(bFlag AND X19 AND M40 AND NOT abComp, bFlagExe);
(* network 3 *)
ZP_BUFRCV(bFlagExe, "U0", 1, aCtrlData, D500, abComp);
(* network 4 *)
SET(abComp[0] AND NOT abComp[1], bNormal);
SET(abComp[0] AND abComp[1], bError);
(* network 5 *)
Z_BUFRCVS(SM400, "U0", 1, D500);
END_PROGRAM

PROGRAM ExBUFSND
(* structured ladder/FBD written out as ST: instructions are called as NAME(EN, inputs, outputs); _pN, _eN, _tN stand for wires *)
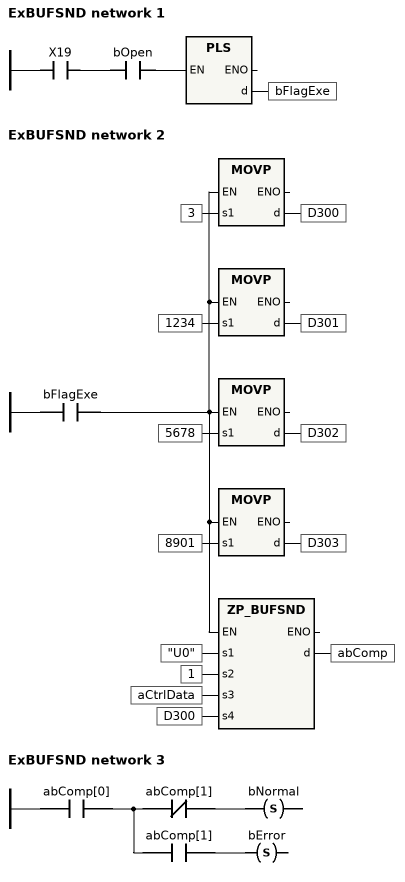
(* network 1 *)
PLS(X19 AND bOpen, bFlagExe);
(* network 2 *)
MOVP(bFlagExe, 3, D300);
MOVP(bFlagExe, 1234, D301);
MOVP(bFlagExe, 5678, D302);
MOVP(bFlagExe, 8901, D303);
ZP_BUFSND(bFlagExe, "U0", 1, aCtrlData, D300, abComp);
(* network 3 *)
SET(abComp[0] AND NOT abComp[1], bNormal);
SET(abComp[0] AND abComp[1], bError);
END_PROGRAM

PROGRAM ExERRCLR
VAR
  bReqFlag : BOOL;
  bFlagExe : BOOL;
  abComp : ARRAY [0..1] OF BOOL;
  aCtrlData : ARRAY [0..7] OF INT;
  iErrCode : INT;
END_VAR
(* structured ladder/FBD written out as ST: instructions are called as NAME(EN, inputs, outputs); _pN, _eN, _tN stand for wires *)
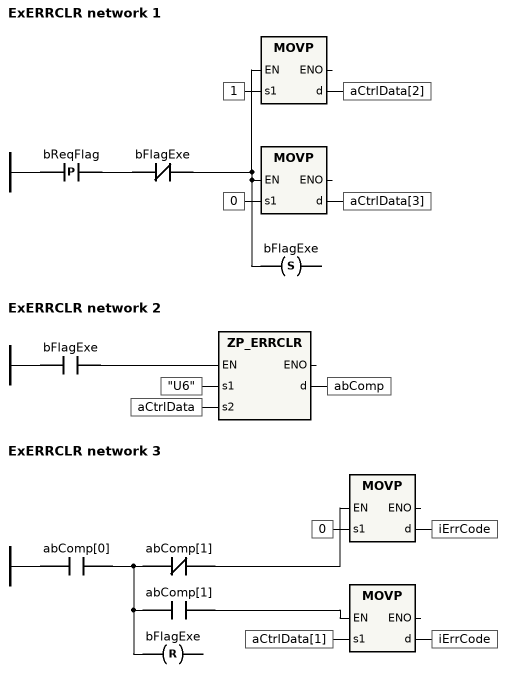
(* network 1 *)
_p1 := LDP(TRUE, bReqFlag) AND NOT bFlagExe;
MOVP(_p1, 1, aCtrlData[2]);
MOVP(_p1, 0, aCtrlData[3]);
SET(_p1, bFlagExe);
(* network 2 *)
ZP_ERRCLR(bFlagExe, "U6", aCtrlData, abComp);
(* network 3 *)
MOVP(abComp[0] AND NOT abComp[1], 0, iErrCode);
MOVP(abComp[0] AND abComp[1], aCtrlData[1], iErrCode);
RST(abComp[0], bFlagExe);
END_PROGRAM

PROGRAM ExMRECV
VAR
  abComp : ARRAY [0..1] OF BOOL;
  Mov4INT_1 : Mov4INT;
  aCtrlData : ARRAY [0..15] OF INT;
  bCmdFlag : BOOL;
  bExeFlag : BOOL;
END_VAR
(* structured ladder/FBD written out as ST: instructions are called as NAME(EN, inputs, outputs); _pN, _eN, _tN stand for wires *)
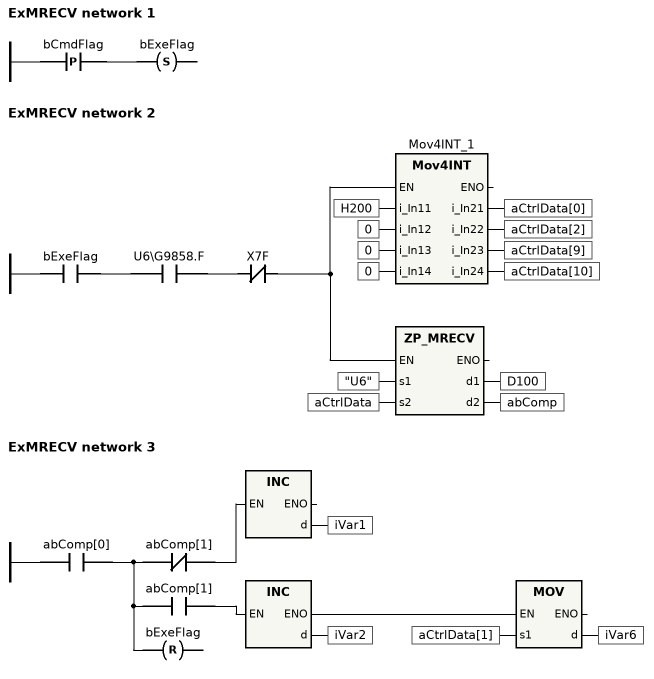
(* network 1 *)
SET(LDP(TRUE, bCmdFlag), bExeFlag);
(* network 2 *)
_p1 := bExeFlag AND U6\G9858.F AND NOT X7F;
Mov4INT_1(EN := _p1, i_In11 := H200, i_In12 := 0, i_In13 := 0, i_In14 := 0, i_In21 => aCtrlData[0], i_In22 => aCtrlData[2], i_In23 => aCtrlData[9], i_In24 => aCtrlData[10]);
ZP_MRECV(_p1, "U6", aCtrlData, D100, abComp);
(* network 3 *)
INC(abComp[0] AND NOT abComp[1], iVar1);
_e1 := INC(abComp[0] AND abComp[1], iVar2);
MOV(_e1, aCtrlData[1], iVar6);
RST(abComp[0], bExeFlag);
END_PROGRAM

PROGRAM ExMSEND
VAR
  abComp : ARRAY [0..1] OF BOOL;
  Mov4INT_1 : Mov4INT;
  aCtrlData : ARRAY [0..15] OF INT;
  bCmdFlag : BOOL;
  bExeFlag : BOOL;
  Mov4INT_2 : Mov4INT;
END_VAR
(* structured ladder/FBD written out as ST: instructions are called as NAME(EN, inputs, outputs); _pN, _eN, _tN stand for wires *)
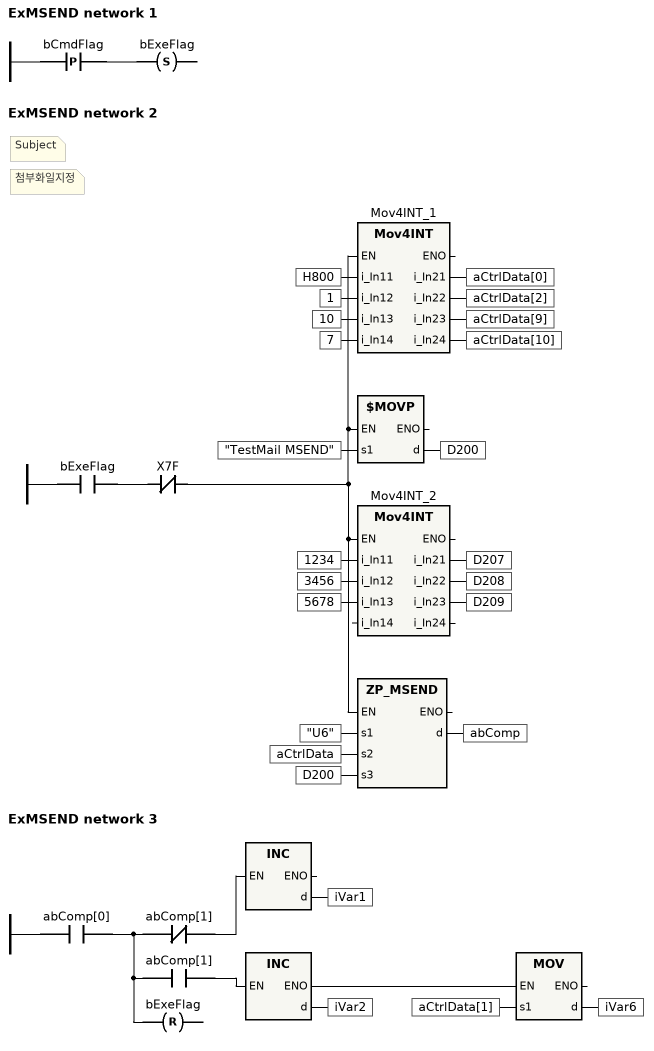
(* network 1 *)
SET(LDP(TRUE, bCmdFlag), bExeFlag);
(* network 2 *)
(* Subject *)
(* 첨부화일지정 *)
_p1 := bExeFlag AND NOT X7F;
Mov4INT_1(EN := _p1, i_In11 := H800, i_In12 := 1, i_In13 := 10, i_In14 := 7, i_In21 => aCtrlData[0], i_In22 => aCtrlData[2], i_In23 => aCtrlData[9], i_In24 => aCtrlData[10]);
$MOVP(_p1, "TestMail MSEND", D200);
Mov4INT_2(EN := _p1, i_In11 := 1234, i_In12 := 3456, i_In13 := 5678, i_In21 => D207, i_In22 => D208, i_In23 => D209);
ZP_MSEND(_p1, "U6", aCtrlData, D200, abComp);
(* network 3 *)
INC(abComp[0] AND NOT abComp[1], iVar1);
_e1 := INC(abComp[0] AND abComp[1], iVar2);
MOV(_e1, aCtrlData[1], iVar6);
RST(abComp[0], bExeFlag);
END_PROGRAM

PROGRAM ExUINI
VAR
  bReqFlag : BOOL;
  bFlagExe : BOOL;
  abComp : ARRAY [0..1] OF BOOL;
  aCtrlData : ARRAY [0..9] OF INT;
  iErrCode : INT;
  bInitExe : BOOL;
  bInitComp : BOOL;
  bInitError : BOOL;
  bInitComp2 : BOOL;
  bInitError2 : BOOL;
  bInitCompEnd : BOOL;
END_VAR
(* structured ladder/FBD written out as ST: instructions are called as NAME(EN, inputs, outputs); _pN, _eN, _tN stand for wires *)
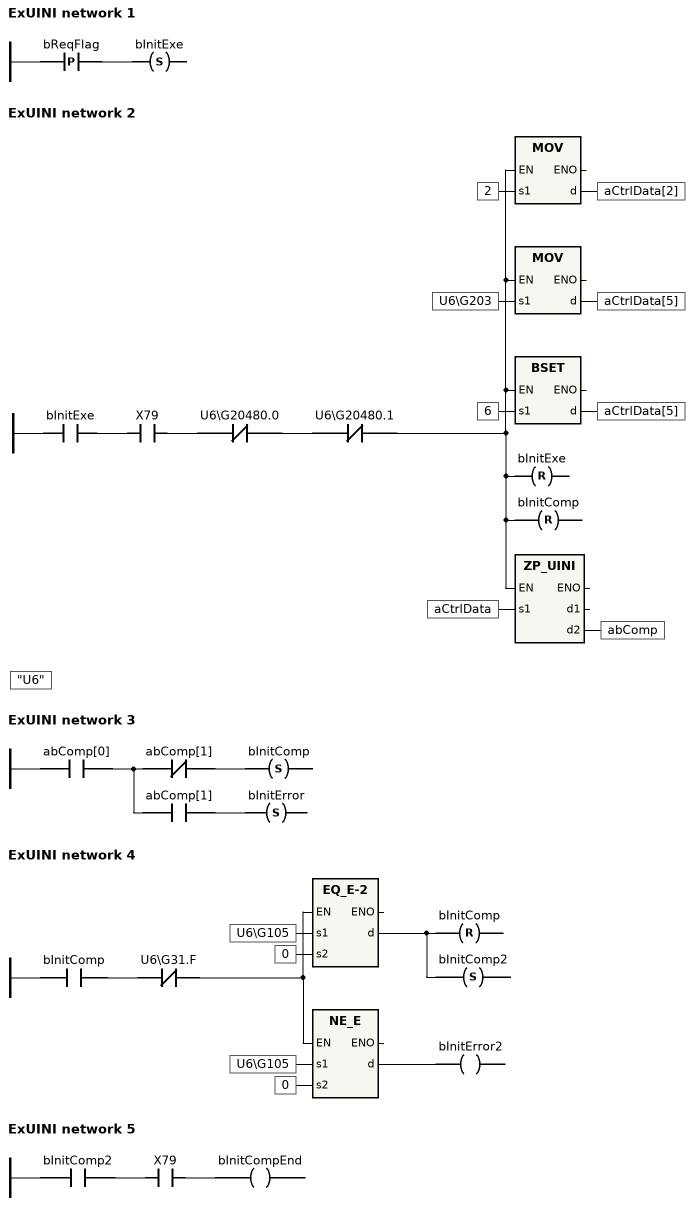
(* network 1 *)
SET(LDP(TRUE, bReqFlag), bInitExe);
(* network 2 *)
_p1 := bInitExe AND X79 AND NOT U6\G20480.0 AND NOT U6\G20480.1;
MOV(_p1, 2, aCtrlData[2]);
MOV(_p1, U6\G203, aCtrlData[5]);
BSET(_p1, 6, aCtrlData[5]);
ZP_UINI(_p1, aCtrlData, _open, abComp);
RST(_p1, bInitExe);
RST(_p1, bInitComp);
(* not connected to any output: "U6" *)
(* network 3 *)
SET(abComp[0] AND NOT abComp[1], bInitComp);
SET(abComp[0] AND abComp[1], bInitError);
(* network 4 *)
_p1 := bInitComp AND NOT U6\G31.F;
EQ_E(_p1, U6\G105, 0, _t2);
RST(_t2, bInitComp);
SET(_t2, bInitComp2);
NE_E(_p1, U6\G105, 0, _t3);
bInitError2 := _t3;
(* network 5 *)
bInitCompEnd := bInitComp2 AND X79;
END_PROGRAM

PROGRAM ExEthREAD_WRITE
VAR
  Mov8INT_1 : Mov8INT;
  acRdCtrl : ARRAY [0..17] OF INT;
  abRdComp : ARRAY [0..1] OF BOOL;
  iCntRdOk : INT;
  iCntRdErr : INT;
  acWrCtrl : ARRAY [0..17] OF INT;
  abWrComp : ARRAY [0..1] OF BOOL;
  Mov8INT_2 : Mov8INT;
  iCntWrOk : INT;
  iCntWrErr : INT;
END_VAR
(* structured ladder/FBD written out as ST: instructions are called as NAME(EN, inputs, outputs); _pN, _eN, _tN stand for wires *)
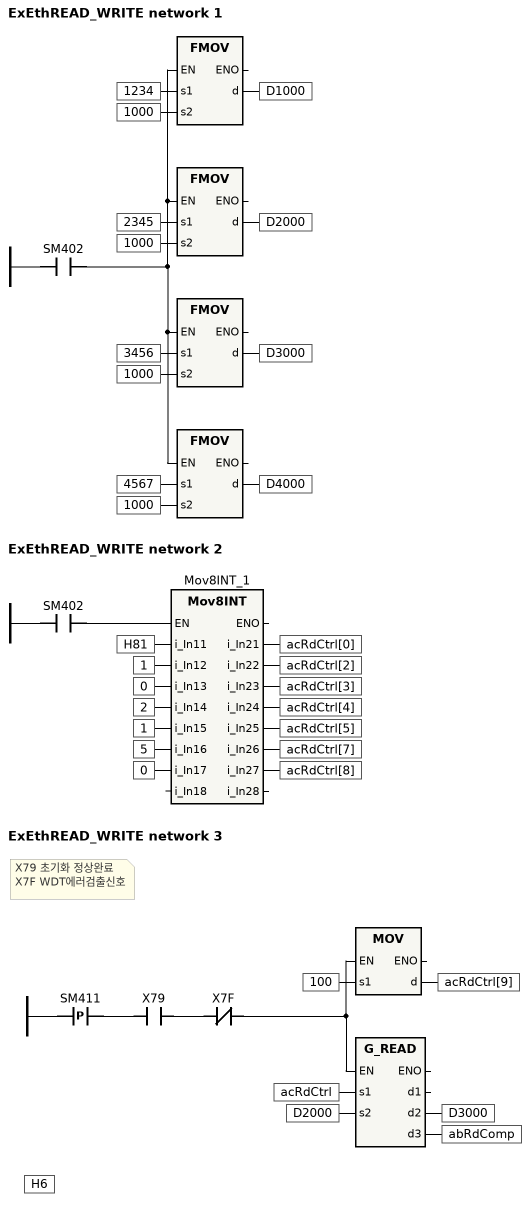
(* network 1 *)
FMOV(SM402, 1234, 1000, D1000);
FMOV(SM402, 2345, 1000, D2000);
FMOV(SM402, 3456, 1000, D3000);
FMOV(SM402, 4567, 1000, D4000);
(* network 2 *)
Mov8INT_1(EN := SM402, i_In11 := H81, i_In12 := 1, i_In13 := 0, i_In14 := 2, i_In15 := 1, i_In16 := 5, i_In17 := 0, i_In21 => acRdCtrl[0], i_In22 => acRdCtrl[2], i_In23 => acRdCtrl[3], i_In24 => acRdCtrl[4], i_In25 => acRdCtrl[5], i_In26 => acRdCtrl[7], i_In27 => acRdCtrl[8]);
(* network 3 *)
(* X79 초기화 정상완료 / X7F WDT에러검출신호 *)
_p1 := LDP(TRUE, SM411) AND X79 AND NOT X7F;
MOV(_p1, 100, acRdCtrl[9]);
G_READ(_p1, acRdCtrl, D2000, _open, D3000, abRdComp);
(* not connected to any output: H6 *)
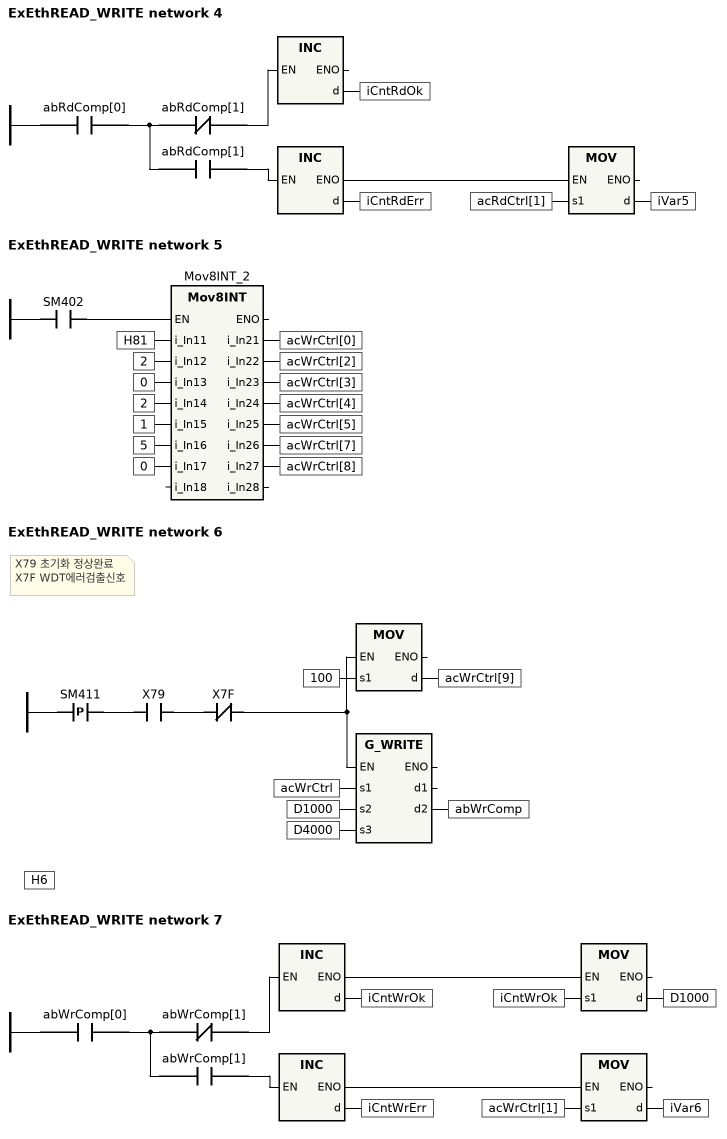
(* network 4 *)
INC(abRdComp[0] AND NOT abRdComp[1], iCntRdOk);
_e1 := INC(abRdComp[0] AND abRdComp[1], iCntRdErr);
MOV(_e1, acRdCtrl[1], iVar5);
(* network 5 *)
Mov8INT_2(EN := SM402, i_In11 := H81, i_In12 := 2, i_In13 := 0, i_In14 := 2, i_In15 := 1, i_In16 := 5, i_In17 := 0, i_In21 => acWrCtrl[0], i_In22 => acWrCtrl[2], i_In23 => acWrCtrl[3], i_In24 => acWrCtrl[4], i_In25 => acWrCtrl[5], i_In26 => acWrCtrl[7], i_In27 => acWrCtrl[8]);
(* network 6 *)
(* X79 초기화 정상완료 / X7F WDT에러검출신호 *)
_p1 := LDP(TRUE, SM411) AND X79 AND NOT X7F;
MOV(_p1, 100, acWrCtrl[9]);
G_WRITE(_p1, acWrCtrl, D1000, D4000, _open, abWrComp);
(* not connected to any output: H6 *)
(* network 7 *)
_e1 := INC(abWrComp[0] AND NOT abWrComp[1], iCntWrOk);
MOV(_e1, iCntWrOk, D1000);
_e2 := INC(abWrComp[0] AND abWrComp[1], iCntWrErr);
MOV(_e2, acWrCtrl[1], iVar6);
END_PROGRAM

FUNCTION_BLOCK Word2Bit8
VAR_INPUT
  IN : WORD;
END_VAR
VAR_OUTPUT
  Bit0 : BOOL;
  Bit1 : BOOL;
  Bit2 : BOOL;
  Bit3 : BOOL;
  Bit4 : BOOL;
  Bit5 : BOOL;
  Bit6 : BOOL;
  Bit7 : BOOL;
END_VAR
 
Bit0 := WORD_TO_BOOL(IN AND 16#0001);
Bit1 := WORD_TO_BOOL(SHR(IN AND 16#0002 , 1));
Bit2 := WORD_TO_BOOL(SHR(IN AND 16#0004 , 2));
Bit3 := WORD_TO_BOOL(SHR(IN AND 16#0008 , 3));
Bit4 := WORD_TO_BOOL(SHR(IN AND 16#0010 , 4));
Bit5 := WORD_TO_BOOL(SHR(IN AND 16#0020 , 5));
Bit6 := WORD_TO_BOOL(SHR(IN AND 16#0040 , 6));
Bit7 := WORD_TO_BOOL(SHR(IN AND 16#0080 , 7));
END_FUNCTION_BLOCK

PROGRAM ExEfullCact
VAR
  bOpenReqC : BOOL;
  bCsetReq : BOOL;
  bOpenReqE : BOOL;
  bOpenOkC : BOOL;
  bOpenOkE : BOOL;
  bOpenErrC : BOOL;
  bOpenErrE : BOOL;
  abOpenResC : ARRAY [0..1] OF BOOL;
  abOpenResE : ARRAY [0..1] OF BOOL;
  acOpenData : ARRAY [0..9] OF INT;
  acCsetData : ARRAY [0..4] OF INT;
  acRdCtrl : ARRAY [0..9] OF INT;
  bSendReqC : BOOL;
  bSendReqE : BOOL;
  bSendOkC : BOOL;
  bSendOkE : BOOL;
  bSendErrC : BOOL;
  bSendErrE : BOOL;
  abSendResC : ARRAY [0..1] OF BOOL;
  abSendResE : ARRAY [0..1] OF BOOL;
  abSendResF : ARRAY [0..1] OF BOOL;
  acSendDataC : ARRAY [0..1] OF INT;
  acSendDataE : ARRAY [0..1] OF INT;
  acSendDataF : ARRAY [0..1] OF INT;
  bRecvOkC : BOOL;
  bRecvOkE : BOOL;
  bRecvOkF : BOOL;
  bRecvErrC : BOOL;
  bRecvErrE : BOOL;
  bRecvErrF : BOOL;
  abRecvResC : ARRAY [0..1] OF BOOL;
  abRecvResE : ARRAY [0..1] OF BOOL;
  abRecvResF : ARRAY [0..1] OF BOOL;
  acRecvDataC : ARRAY [0..1] OF INT;
  acRecvDataE : ARRAY [0..1] OF INT;
  acRecvDataF : ARRAY [0..1] OF INT;
  bCloseReq : BOOL;
  bCloseOkC : BOOL;
  bCloseOkE : BOOL;
  bCloseErrC : BOOL;
  bCloseErrE : BOOL;
  abCloseResC : ARRAY [0..1] OF BOOL;
  abCloseResE : ARRAY [0..1] OF BOOL;
  acCloseData : ARRAY [0..1] OF INT;
  CntSend1 : INT;
  CntSend2 : INT;
  CntSend3 : INT;
  CntRecv1 : INT;
  CntRecvErr1 : INT;
  CntRecv2 : INT;
  CntRecv3 : INT;
  CntRecvErr2 : INT;
  CntRecvErr3 : INT;
  ErrCodeSC : INT;
  ErrCodeSE : INT;
  ErrCodeSF : INT;
  ErrCodeRC : INT;
  ErrCodeRE : INT;
  ErrCodeRF : INT;
  Mov4INT_1 : Mov4INT;
  Mov8INT_1 : Mov8INT;
  Mov4INT_2 : Mov4INT;
  Mov4INT_3 : Mov4INT;
  Mov4INT_4 : Mov4INT;
  Word2Bit8_1 : Word2Bit8;
  Word2Bit8_2 : Word2Bit8;
  Word2Bit8_3 : Word2Bit8;
  Word2Bit8_4 : Word2Bit8;
  Word2Bit8_5 : Word2Bit8;
  Word2Bit8_6 : Word2Bit8;
  TON_1 : TON;
  TON_2 : TON;
  TON_3 : TON;
END_VAR
(* structured ladder/FBD written out as ST: instructions are called as NAME(EN, inputs, outputs); _pN, _eN, _tN stand for wires *)
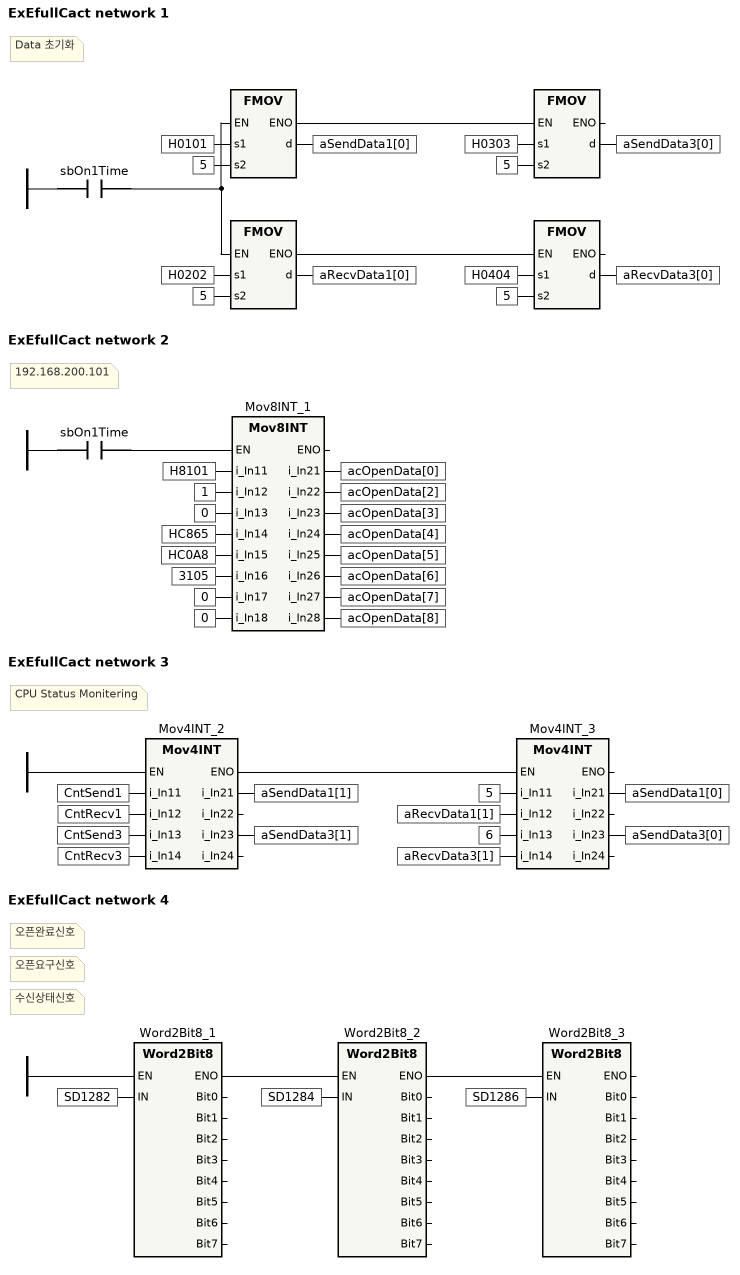
(* network 1 *)
(* Data 초기화 *)
_e1 := FMOV(sbOn1Time, H0101, 5, aSendData1[0]);
FMOV(_e1, H0303, 5, aSendData3[0]);
_e2 := FMOV(sbOn1Time, H0202, 5, aRecvData1[0]);
FMOV(_e2, H0404, 5, aRecvData3[0]);
(* network 2 *)
(* 192.168.200.101 *)
Mov8INT_1(EN := sbOn1Time, i_In11 := H8101, i_In12 := 1, i_In13 := 0, i_In14 := HC865, i_In15 := HC0A8, i_In16 := 3105, i_In17 := 0, i_In18 := 0, i_In21 => acOpenData[0], i_In22 => acOpenData[2], i_In23 => acOpenData[3], i_In24 => acOpenData[4], i_In25 => acOpenData[5], i_In26 => acOpenData[6], i_In27 => acOpenData[7], i_In28 => acOpenData[8]);
(* network 3 *)
(* CPU Status Monitering *)
Mov4INT_2(EN := TRUE, i_In11 := CntSend1, i_In12 := CntRecv1, i_In13 := CntSend3, i_In14 := CntRecv3, i_In21 => aSendData1[1], i_In23 => aSendData3[1]);
Mov4INT_3(EN := Mov4INT_2.ENO, i_In11 := 5, i_In12 := aRecvData1[1], i_In13 := 6, i_In14 := aRecvData3[1], i_In21 => aSendData1[0], i_In23 => aSendData3[0]);
(* network 4 *)
(* 오픈완료신호 *)
(* 오픈요구신호 *)
(* 수신상태신호 *)
Word2Bit8_1(EN := TRUE, IN := SD1282);
Word2Bit8_2(EN := Word2Bit8_1.ENO, IN := SD1284);
Word2Bit8_3(EN := Word2Bit8_2.ENO, IN := SD1286);
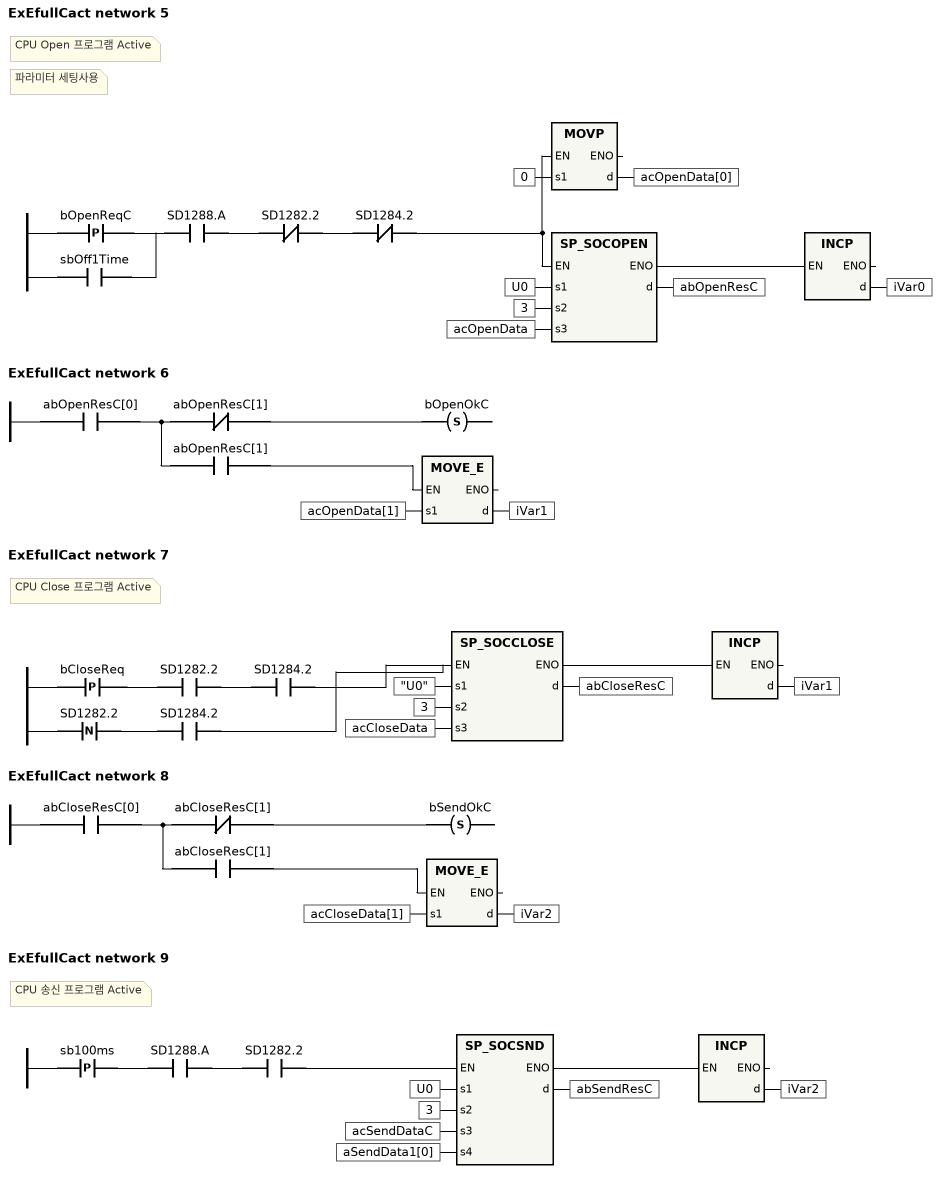
(* network 5 *)
(* CPU Open 프로그램 Active *)
(* 파라미터 세팅사용 *)
_p1 := (((LDP(TRUE, bOpenReqC) OR sbOff1Time) AND SD1288.A) AND NOT SD1282.2) AND NOT SD1284.2;
MOVP(_p1, 0, acOpenData[0]);
_e2 := SP_SOCOPEN(_p1, U0, 3, acOpenData, abOpenResC);
INCP(_e2, iVar0);
(* network 6 *)
SET(abOpenResC[0] AND NOT abOpenResC[1], bOpenOkC);
MOVE_E(abOpenResC[0] AND abOpenResC[1], acOpenData[1], iVar1);
(* network 7 *)
(* CPU Close 프로그램 Active *)
_e1 := SP_SOCCLOSE((LDP(TRUE, bCloseReq) AND SD1282.2 AND SD1284.2) OR (LDF(TRUE, SD1282.2) AND SD1284.2), "U0", 3, acCloseData, abCloseResC);
INCP(_e1, iVar1);
(* network 8 *)
SET(abCloseResC[0] AND NOT abCloseResC[1], bSendOkC);
MOVE_E(abCloseResC[0] AND abCloseResC[1], acCloseData[1], iVar2);
(* network 9 *)
(* CPU 송신 프로그램 Active *)
_e1 := SP_SOCSND(LDP(TRUE, sb100ms) AND SD1288.A AND SD1282.2, U0, 3, acSendDataC, aSendData1[0], abSendResC);
INCP(_e1, iVar2);
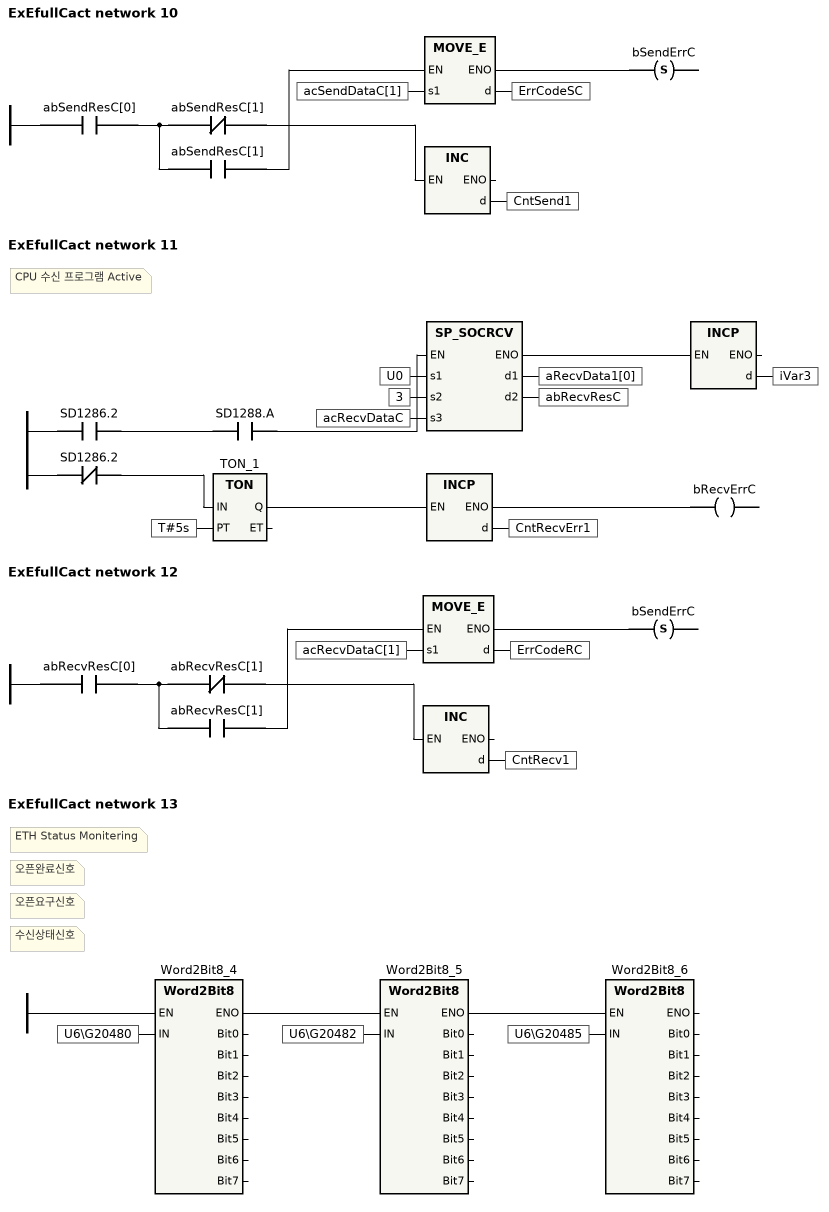
(* network 10 *)
INC(abSendResC[0] AND NOT abSendResC[1], CntSend1);
_e1 := MOVE_E(abSendResC[0] AND abSendResC[1], acSendDataC[1], ErrCodeSC);
SET(_e1, bSendErrC);
(* network 11 *)
(* CPU 수신 프로그램 Active *)
_e1 := SP_SOCRCV(SD1286.2 AND SD1288.A, U0, 3, acRecvDataC, aRecvData1[0], abRecvResC);
INCP(_e1, iVar3);
TON_1(IN := NOT SD1286.2, PT := T#5s);
_e2 := INCP(TON_1.Q, CntRecvErr1);
bRecvErrC := _e2;
(* network 12 *)
INC(abRecvResC[0] AND NOT abRecvResC[1], CntRecv1);
_e1 := MOVE_E(abRecvResC[0] AND abRecvResC[1], acRecvDataC[1], ErrCodeRC);
SET(_e1, bSendErrC);
(* network 13 *)
(* ETH Status Monitering *)
(* 오픈완료신호 *)
(* 오픈요구신호 *)
(* 수신상태신호 *)
Word2Bit8_4(EN := TRUE, IN := U6\G20480);
Word2Bit8_5(EN := Word2Bit8_4.ENO, IN := U6\G20482);
Word2Bit8_6(EN := Word2Bit8_5.ENO, IN := U6\G20485);
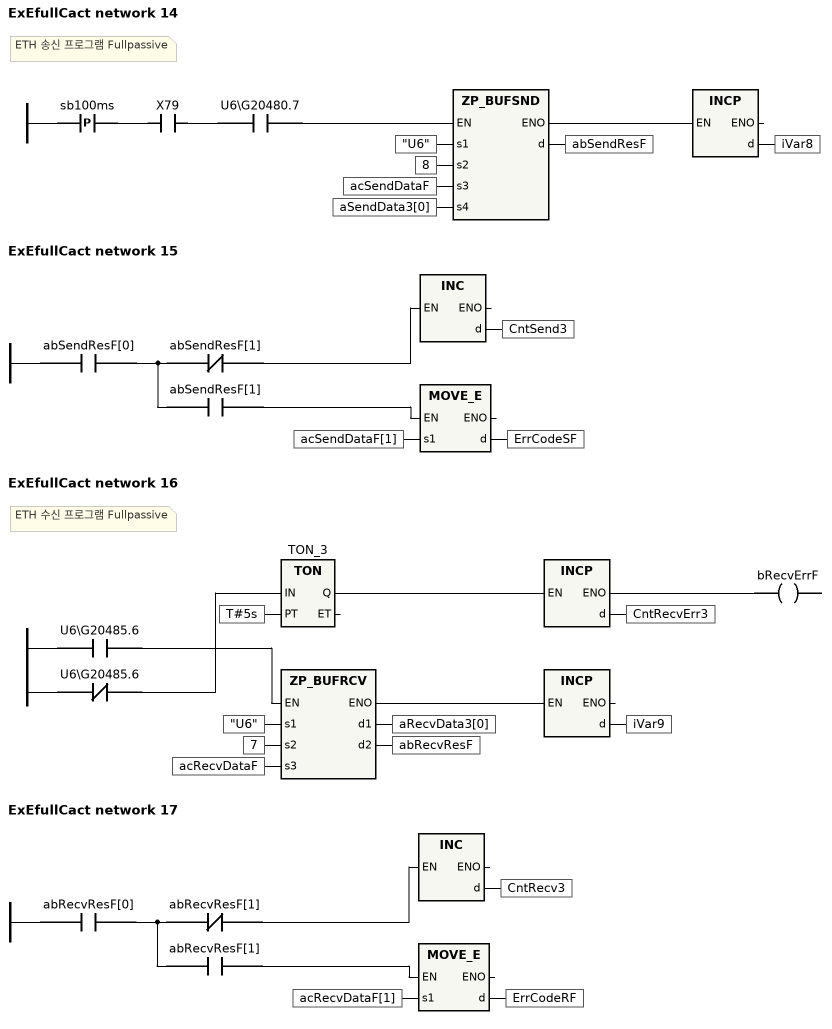
(* network 14 *)
(* ETH 송신 프로그램 Fullpassive *)
_e1 := ZP_BUFSND(LDP(TRUE, sb100ms) AND X79 AND U6\G20480.7, "U6", 8, acSendDataF, aSendData3[0], abSendResF);
INCP(_e1, iVar8);
(* network 15 *)
INC(abSendResF[0] AND NOT abSendResF[1], CntSend3);
MOVE_E(abSendResF[0] AND abSendResF[1], acSendDataF[1], ErrCodeSF);
(* network 16 *)
(* ETH 수신 프로그램 Fullpassive *)
_e1 := ZP_BUFRCV(U6\G20485.6, "U6", 7, acRecvDataF, aRecvData3[0], abRecvResF);
INCP(_e1, iVar9);
TON_3(IN := NOT U6\G20485.6, PT := T#5s);
_e2 := INCP(TON_3.Q, CntRecvErr3);
bRecvErrF := _e2;
(* network 17 *)
INC(abRecvResF[0] AND NOT abRecvResF[1], CntRecv3);
MOVE_E(abRecvResF[0] AND abRecvResF[1], acRecvDataF[1], ErrCodeRF);
END_PROGRAM

PROGRAM ExEactCact
VAR
  bOpenReqC : BOOL;
  bOpenOkC : BOOL;
  bOpenErrC : BOOL;
  abOpenResC : ARRAY [0..1] OF BOOL;
  acOpenDataC : ARRAY [0..9] OF INT;
  bSendReqC : BOOL;
  bSendOkC : BOOL;
  bSendErrC : BOOL;
  abSendResC : ARRAY [0..1] OF BOOL;
  acSendDataC : ARRAY [0..1] OF INT;
  bRecvOkC : BOOL;
  bRecvErrC : BOOL;
  abRecvResC : ARRAY [0..1] OF BOOL;
  bCloseReqC : BOOL;
  bCloseOkC : BOOL;
  bCloseErrC : BOOL;
  abCloseResC : ARRAY [0..1] OF BOOL;
  acCloseDataC : ARRAY [0..1] OF INT;
  CntSend1 : INT;
  CntSend2 : INT;
  CntRecv1 : INT;
  CntRecv2 : INT;
  Mov4INT_1 : Mov4INT;
  Mov8INT_1 : Mov8INT;
  acRdCtrl : ARRAY [0..9] OF INT;
  Mov4INT_2 : Mov4INT;
  bOpenReqE : BOOL;
  bOpenOkE : BOOL;
  bOpenErrE : BOOL;
  abOpenResE : ARRAY [0..1] OF BOOL;
  bSendErrE : BOOL;
  bSendOkE : BOOL;
  bSendReqE : BOOL;
  abSendResE : ARRAY [0..1] OF BOOL;
  abRecvResE : ARRAY [0..1] OF BOOL;
  bRecvErrE : BOOL;
  bRecvOkE : BOOL;
  abCloseResE : ARRAY [0..1] OF BOOL;
  bCloseErrE : BOOL;
  bCloseOkE : BOOL;
  acSendDataE : ARRAY [0..1] OF INT;
  acRecvDataC : ARRAY [0..1] OF INT;
  acRecvDataE : ARRAY [0..1] OF INT;
  Word2Bit8_1 : Word2Bit8;
  Word2Bit8_2 : Word2Bit8;
  Word2Bit8_3 : Word2Bit8;
  Word2Bit8_4 : Word2Bit8;
  Word2Bit8_5 : Word2Bit8;
  Word2Bit8_6 : Word2Bit8;
  ErrCodeSC : INT;
  ErrCodeSE : INT;
  Mov4INT_3 : Mov4INT;
  bChangeReqC : BOOL;
  Mov4INT_4 : Mov4INT;
  acCsetData : ARRAY [0..4] OF INT;
  TON_1 : TON;
  CntRecvErr1 : INT;
  CntRecvErr2 : INT;
  TON_2 : TON;
  ErrCodeRC : INT;
  ErrCodeRE : INT;
  bCloseReqE : BOOL;
  acOpenDataE : ARRAY [0..9] OF INT;
  acCloseDataE : ARRAY [0..1] OF INT;
END_VAR
(* structured ladder/FBD written out as ST: instructions are called as NAME(EN, inputs, outputs); _pN, _eN, _tN stand for wires *)
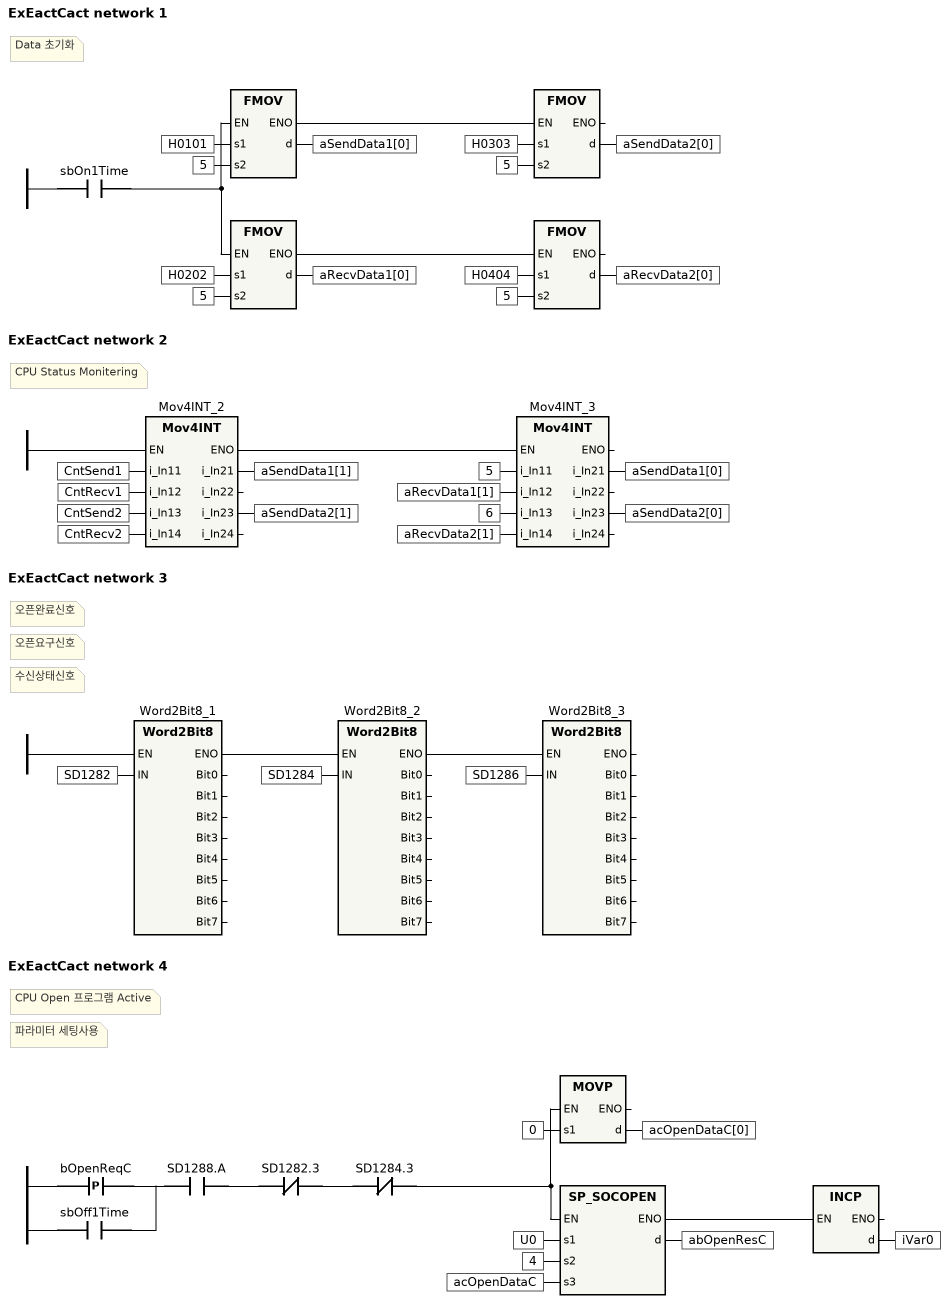
(* network 1 *)
(* Data 초기화 *)
_e1 := FMOV(sbOn1Time, H0101, 5, aSendData1[0]);
FMOV(_e1, H0303, 5, aSendData2[0]);
_e2 := FMOV(sbOn1Time, H0202, 5, aRecvData1[0]);
FMOV(_e2, H0404, 5, aRecvData2[0]);
(* network 2 *)
(* CPU Status Monitering *)
Mov4INT_2(EN := TRUE, i_In11 := CntSend1, i_In12 := CntRecv1, i_In13 := CntSend2, i_In14 := CntRecv2, i_In21 => aSendData1[1], i_In23 => aSendData2[1]);
Mov4INT_3(EN := Mov4INT_2.ENO, i_In11 := 5, i_In12 := aRecvData1[1], i_In13 := 6, i_In14 := aRecvData2[1], i_In21 => aSendData1[0], i_In23 => aSendData2[0]);
(* network 3 *)
(* 오픈완료신호 *)
(* 오픈요구신호 *)
(* 수신상태신호 *)
Word2Bit8_1(EN := TRUE, IN := SD1282);
Word2Bit8_2(EN := Word2Bit8_1.ENO, IN := SD1284);
Word2Bit8_3(EN := Word2Bit8_2.ENO, IN := SD1286);
(* network 4 *)
(* CPU Open 프로그램 Active *)
(* 파라미터 세팅사용 *)
_p1 := (((LDP(TRUE, bOpenReqC) OR sbOff1Time) AND SD1288.A) AND NOT SD1282.3) AND NOT SD1284.3;
MOVP(_p1, 0, acOpenDataC[0]);
_e2 := SP_SOCOPEN(_p1, U0, 4, acOpenDataC, abOpenResC);
INCP(_e2, iVar0);
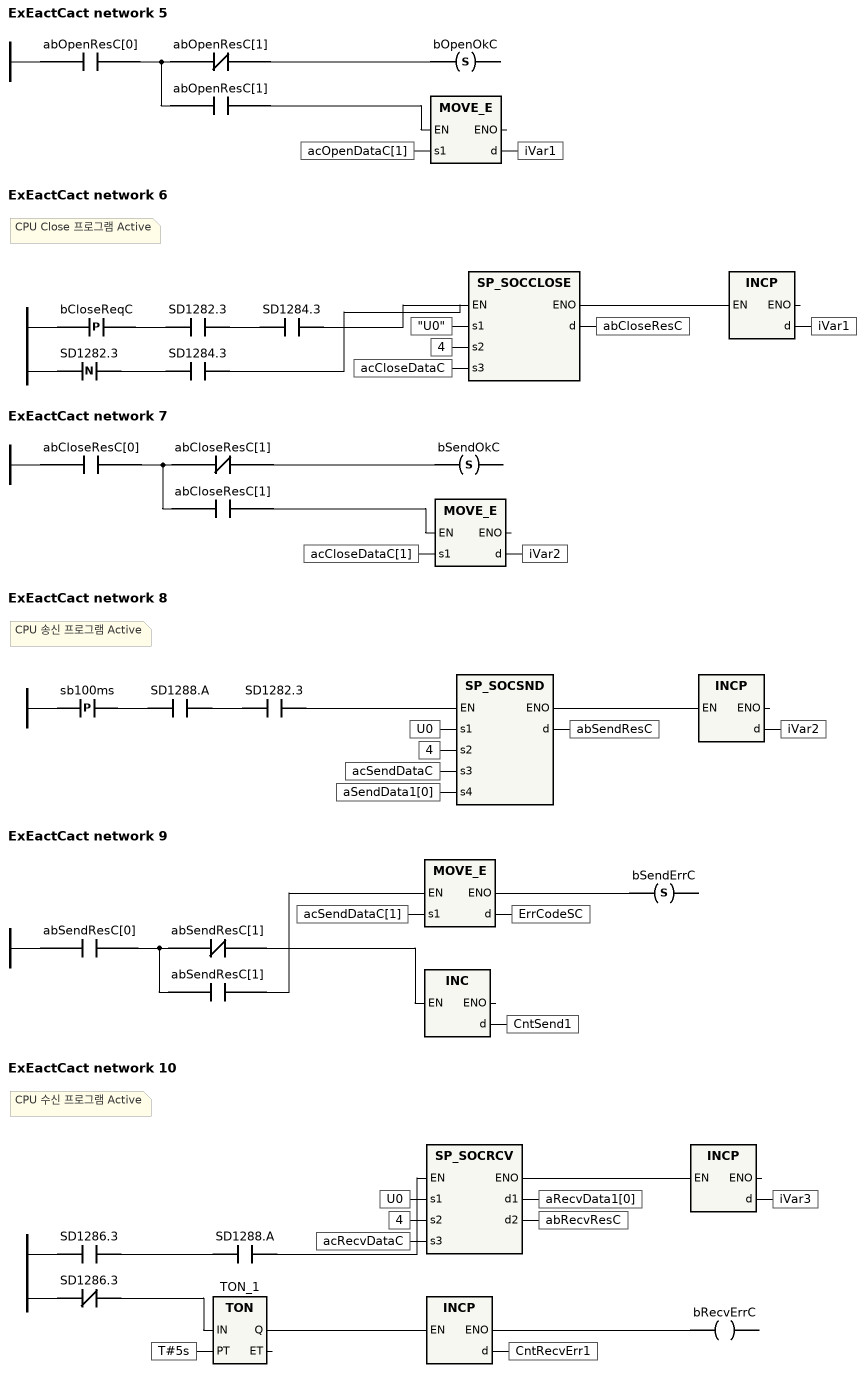
(* network 5 *)
SET(abOpenResC[0] AND NOT abOpenResC[1], bOpenOkC);
MOVE_E(abOpenResC[0] AND abOpenResC[1], acOpenDataC[1], iVar1);
(* network 6 *)
(* CPU Close 프로그램 Active *)
_e1 := SP_SOCCLOSE((LDP(TRUE, bCloseReqC) AND SD1282.3 AND SD1284.3) OR (LDF(TRUE, SD1282.3) AND SD1284.3), "U0", 4, acCloseDataC, abCloseResC);
INCP(_e1, iVar1);
(* network 7 *)
SET(abCloseResC[0] AND NOT abCloseResC[1], bSendOkC);
MOVE_E(abCloseResC[0] AND abCloseResC[1], acCloseDataC[1], iVar2);
(* network 8 *)
(* CPU 송신 프로그램 Active *)
_e1 := SP_SOCSND(LDP(TRUE, sb100ms) AND SD1288.A AND SD1282.3, U0, 4, acSendDataC, aSendData1[0], abSendResC);
INCP(_e1, iVar2);
(* network 9 *)
INC(abSendResC[0] AND NOT abSendResC[1], CntSend1);
_e1 := MOVE_E(abSendResC[0] AND abSendResC[1], acSendDataC[1], ErrCodeSC);
SET(_e1, bSendErrC);
(* network 10 *)
(* CPU 수신 프로그램 Active *)
_e1 := SP_SOCRCV(SD1286.3 AND SD1288.A, U0, 4, acRecvDataC, aRecvData1[0], abRecvResC);
INCP(_e1, iVar3);
TON_1(IN := NOT SD1286.3, PT := T#5s);
_e2 := INCP(TON_1.Q, CntRecvErr1);
bRecvErrC := _e2;
